FOR nIdxScan := 1 TO nNumberOfSensors DO
	//Setup parameters
		//Setup Motion part of sensor (Instance 0)
		arrNiko_P46xx[nIdxScan].eEventPriorityOccupancy:= stSensorSetup.eEventPriorityOccupancy;
		arrNiko_P46xx[nIdxScan].nHoldTimerOccupancy := stSensorSetup.nHoldTimerOccupancy ;
		arrNiko_P46xx[nIdxScan].nReportTimerOccupancy := stSensorSetup.nReportTimerOccupancy;
		arrNiko_P46xx[nIdxScan].nDeadtimeTimerOccupancy:= stSensorSetup.nDeadtimeTimerOccupancy;
		arrNiko_P46xx[nIdxScan].nSensitivityOccupancyA:= stSensorSetup.nSensitivityPIRSegmentA;
		arrNiko_P46xx[nIdxScan].nSensitivityOccupancyB:= stSensorSetup.nSensitivityPIRSegmentB;
		arrNiko_P46xx[nIdxScan].nSensitivityOccupancyC:= stSensorSetup.nSensitivityPIRSegmentC;
	
		//Setup Brightness part of sensor (Instance 1)
		arrNiko_P46xx[nIdxScan].bEnableBrightness := stSensorSetup.bEnableInstanceBrightness;
		arrNiko_P46xx[nIdxScan].eEventPriorityBrightness:= stSensorSetup.eEventPriorityBrightness;
		arrNiko_P46xx[nIdxScan].nDeadtimeTimerBrightness:= stSensorSetup.nDeadtimeTimerBrightness;
		arrNiko_P46xx[nIdxScan].nHysteresisBrightness:= stSensorSetup.nHysteresisBrightness;
		arrNiko_P46xx[nIdxScan].nHysteresisMinBrightness:= stSensorSetup.nHysteresisMinBrightness;
		arrNiko_P46xx[nIdxScan].nReportTimerBrightness:= stSensorSetup.nReportTimerBrightness;
		
	//Calculate delay time for init sensor
	arrtDelayTime[nIdxScan] := INT_TO_TIME((BYTE_TO_INT(arrShrtAdr[nIdxScan]) * 400));	
	arrDelaySetupDALIDevice[nIdxScan](IN:= bInitialize , PT:=arrtDelayTime[nIdxScan] , Q=> , ET=> );	
		
	IF arrDelaySetupDALIDevice[nIdxScan].q AND NOT GVL_DALI.arrbBlockDTR[DALI_LINE_NUM] AND NOT (arrInitDone[nIdxScan] OR arrInitErr[nIdxScan]) THEN
		arrInitSensor[nIdxScan]:= TRUE;
		GVL_DALI.arrbBlockDTR[DALI_LINE_NUM]:= TRUE;
	END_IF
	
	bQueryBrightness:= stPirSensorData.bQueryBrightness OR NOT bAutoRead;
	
	fbAutoRequestBrightness_TON(IN:= NOT fbAutoRequestBrightness_TON.Q  AND NOT stPirSensorData.bQueryBrightness , PT:= (arrtDelayTime[nIdxScan] + T#12M) , Q=>bAutoRead , ET=> );
	
	bQueryOccupancy:= NOT bAutoRead OR stPirSensorData.bQueryBrightness;
	
	arrNiko_P46xx[nIdxScan](
		bError=> , 
		ipResultMessage=> , 
		bInitialize:=  arrInitSensor[nIdxScan], 
		nShortAddress:= arrShrtAdr[nIdxScan], 
		nOptions:= , 
		bQueryOccupancy:= bQueryOccupancy, 
		bQueryBrightness:= bQueryBrightness, 
		bCancelHoldTimerOccupancy:= bCancelHoldTimerOccupancy, 
		bInitializing=> arrInitializing[nIdxScan] , 
		bReadingOccupancy=> , 
		bReadingBrightness=> , 
		bOccupied=> , 
		nBrightnessLevel=> );
	
	IF arrNiko_P46xx[nIdxScan].bError THEN
		GVL_DALI_LatestError.arrLineShrtAddr[DALI_LINE_NUM] :=arrShrtAdr[nIdxScan];
	END_IF
	
	arrInitDone_FTrig[nIdxScan](CLK:=arrInitializing[nIdxScan] );	
		IF arrInitDone_FTrig[nIdxScan].Q THEN
			IF NOT bInitTimeOut THEN
				arrInitDone[nIdxScan] := TRUE;
				GVL_DALI.arrbBlockDTR[DALI_LINE_NUM]:= FALSE;
			ELSE
				arrInitErr[nIdxScan] := TRUE;
				GVL_DALI.arrbBlockDTR[DALI_LINE_NUM]:= FALSE;
			END_IF
		END_IF
		
	fbInitTimeOut[nIdxScan](IN:=arrInitSensor[nIdxScan] AND NOT arrInitDone[nIdxScan], PT:= T#10S); 
	
	IF fbInitTimeOut[nIdxScan].Q THEN
		arrInitErr[nIdxScan] := TRUE;
		GVL_DALI.arrbBlockDTR[DALI_LINE_NUM]:= FALSE;
	END_IF
END_FOR

stPirSensorData.bPrc:= FALSE;
FOR nPirIdxOn:= 1 TO nNumberOfSensors DO
	IF arrNiko_P46xx[nPirIdxOn].bOccupied THEN
		stPirSensorData.bPrc:= TRUE;
		EXIT;
	END_IF
END_FOR

stPirSensorData.bBrightnessRead:=	arrNiko_P46xx[1].bReadingBrightness OR arrNiko_P46xx[2].bReadingBrightness OR arrNiko_P46xx[3].bReadingBrightness OR arrNiko_P46xx[4].bReadingBrightness OR arrNiko_P46xx[5].bReadingBrightness OR
														arrNiko_P46xx[6].bReadingBrightness OR arrNiko_P46xx[7].bReadingBrightness OR arrNiko_P46xx[8].bReadingBrightness OR arrNiko_P46xx[9].bReadingBrightness;

fBrightness_1:= F_fScale(0, arrSensorScales[1].fReadMaxSensor, 0, arrSensorScales[1].fMeassureMaxSensor, 0, arrNiko_P46xx[1].nBrightnessLevel);
fBrightness_2:= F_fScale(0, arrSensorScales[2].fReadMaxSensor, 0, arrSensorScales[2].fMeassureMaxSensor, 0, arrNiko_P46xx[2].nBrightnessLevel);
fBrightness_3:= F_fScale(0, arrSensorScales[3].fReadMaxSensor, 0, arrSensorScales[3].fMeassureMaxSensor, 0, arrNiko_P46xx[3].nBrightnessLevel);
fBrightness_4:= F_fScale(0, arrSensorScales[4].fReadMaxSensor, 0, arrSensorScales[4].fMeassureMaxSensor, 0, arrNiko_P46xx[4].nBrightnessLevel);
fBrightness_5:= F_fScale(0, arrSensorScales[5].fReadMaxSensor, 0, arrSensorScales[5].fMeassureMaxSensor, 0, arrNiko_P46xx[5].nBrightnessLevel);
fBrightness_6:= F_fScale(0, arrSensorScales[6].fReadMaxSensor, 0, arrSensorScales[6].fMeassureMaxSensor, 0, arrNiko_P46xx[6].nBrightnessLevel);
fBrightness_7:= F_fScale(0, arrSensorScales[7].fReadMaxSensor, 0, arrSensorScales[7].fMeassureMaxSensor, 0, arrNiko_P46xx[7].nBrightnessLevel);
fBrightness_8:= F_fScale(0, arrSensorScales[8].fReadMaxSensor, 0, arrSensorScales[8].fMeassureMaxSensor, 0, arrNiko_P46xx[8].nBrightnessLevel);
fBrightness_9:= F_fScale(0, arrSensorScales[9].fReadMaxSensor, 0, arrSensorScales[9].fMeassureMaxSensor, 0, arrNiko_P46xx[9].nBrightnessLevel);

IF fBrightness_1 <> 0 THEN
	stPirSensorData.fBrightness:= fBrightness_1;
END_IF
IF fBrightness_2 <> 0 THEN
	stPirSensorData.fBrightness:= MIN(fBrightness_2, stPirSensorData.fBrightness);
END_IF
IF fBrightness_3 <> 0 THEN
	stPirSensorData.fBrightness:=  MIN(fBrightness_3, stPirSensorData.fBrightness);
END_IF
IF fBrightness_4 <> 0 THEN
	stPirSensorData.fBrightness:=  MIN(fBrightness_4, stPirSensorData.fBrightness);
END_IF
IF fBrightness_5 <> 0 THEN
	stPirSensorData.fBrightness:=  MIN(fBrightness_5, stPirSensorData.fBrightness);
END_IF
IF fBrightness_6 <> 0 THEN
	stPirSensorData.fBrightness:= MIN(fBrightness_6, stPirSensorData.fBrightness);
END_IF
IF fBrightness_7 <> 0 THEN
	stPirSensorData.fBrightness:=  MIN(fBrightness_7, stPirSensorData.fBrightness);
END_IF
IF fBrightness_8 <> 0 THEN
	stPirSensorData.fBrightness:=  MIN(fBrightness_8, stPirSensorData.fBrightness);
END_IF
IF fBrightness_9 <> 0 THEN
	stPirSensorData.fBrightness:=  MIN(fBrightness_9, stPirSensorData.fBrightness);
END_IF


IF NOT bInitialize THEN
	FOR nIdxScan := 1 TO nNumberOfSensors DO
		fbInitTimeOut[nIdxScan](IN:= FALSE);
		arrInitDone[nIdxScan] := FALSE;
		arrInitErr[nIdxScan] := FALSE;
	END_FOR
END_IF
END_ACTION

END_FUNCTION_BLOCK

// POUs/DALI/FBs/FB_Short
FUNCTION_BLOCK INTERNAL FB_Short
VAR_INPUT
END_VAR
VAR_OUTPUT
END_VAR
VAR
END_VAR

END_FUNCTION_BLOCK

// POUs/DALI/FBs/FB_ValTrig_F
FUNCTION_BLOCK FB_ValTrig_F
VAR_INPUT
END_VAR
VAR_OUTPUT
END_VAR
VAR
END_VAR

END_FUNCTION_BLOCK

// POUs/DALI/FUNs/F_lrScale_EX
FUNCTION F_lrScale_EX : LREAL
VAR_INPUT
	fX0, fX1, fY0, fY1, fOffset : REAL;
	lrSetValDct					: REAL;
	bEnaLim 					: BOOL;
END_VAR
VAR
	fDeltaY						: REAL;
	fDeltaX						: REAL;
END_VAR

fDeltaY:= fY1-fY0;
fDeltaX :=fX1-fX0;

IF fDeltaX <=0 THEN
	fDeltaX:=1;
END_IF

IF bEnaLim THEN
	F_lrScale_EX:= LIMIT(fY0, REAL_TO_LREAL( (fDeltaY / fDeltaX) * lrSetValDct + fOffset), fY1);
ELSE
	F_lrScale_EX:= REAL_TO_LREAL( (fDeltaY / fDeltaX) * lrSetValDct + fOffset);
END_IF

END_FUNCTION

// POUs/DALI/MUX/Timing/FB_MinOnMinOffTime
FUNCTION_BLOCK  FB_MinOnMinOffTime
VAR
	nIdx: INT;
	fbTon: TON;
END_VAR
VAR_INPUT
	bRunCMD: BOOL;
	bStopCMD : BOOL;
	tMinOnTime: TIME;
	tMinOffTime: TIME;
END_VAR
VAR_OUTPUT
	bOut_Run: BOOL;
	bOut_Stop: BOOL;
END_VAR

CASE nIdx OF

0: (*Init Step*)

bOut_Run:= FALSE;
bOut_Stop:= FALSE;
fbTon(IN:=FALSE);

IF bRunCMD THEN
	nIdx := nIdx + 1;
END_IF

1: (*Check min on Time*)

fbTon(IN:= TRUE, PT:= tMinOnTime , Q=> , ET=> );
bOut_Run:= TRUE;

IF fbTon.Q THEN
	nIdx := nIdx + 1;
END_IF

2: (*Kørsel OK*)

fbTon(IN:= FALSE);

IF bStopCMD THEN
	bOut_Stop:= TRUE;
	bOut_Run:= FALSE;
	nIdx := nIdx + 1;
END_IF

3: (*Check Min Off tiden*)

fbTon(IN:= TRUE, PT:= tMinOffTime , Q=> , ET=> );

IF fbTon.Q THEN
	nIdx := 0;
END_IF






















ELSE
	nIdx := 0;

END_CASE

END_FUNCTION_BLOCK

// POUs/DALI/Operators/FB_BA_Swi
FUNCTION_BLOCK FB_BA_Swi
VAR_INPUT
	bOn : BOOL;
	bOff : BOOL;
	bToggle : BOOL;
END_VAR
VAR_OUTPUT
	bLgt: BOOL;
END_VAR
VAR
	fbOn_RTrig: R_TRIG;
	fbOff_RTrig: R_TRIG;
	fbTogle_RTrig: R_TRIG;

END_VAR


fbOn_RTrig(CLK:= bOn );
fbOff_RTrig(CLK:= bOn );
fbTogle_RTrig(CLK:= bOn );

IF fbOn_RTrig.Q THEN
	bLgt := TRUE;
END_IF

IF fbOff_RTrig.Q THEN
	bLgt := FALSE;
END_IF

IF fbTogle_RTrig.Q THEN
	bLgt := NOT bLgt;
END_IF

END_FUNCTION_BLOCK

// POUs/DALI/Operators/FB_Click
FUNCTION_BLOCK FB_Click
VAR_INPUT
	bSwitch						:	BOOL; (* Input signal. *)
	tSwitchTime					:	TIME := T#50MS; (* Kontrol af længde på tryk *)
END_VAR
VAR_OUTPUT
	bShortClick					:	BOOL; (* Kort tryk indikering *)
	bLongClick					:	BOOL; (* Lang tryk indikering *)
END_VAR
VAR
	fbTimerDelay_TON			:	TON;
	fbRisingEdgeSwitch			:	R_TRIG;
	fbFallingEdgeSwitch			:	F_TRIG;
	bDelayOver					:	BOOL := FALSE;
END_VAR

bShortClick := FALSE;
bLongClick := FALSE;

fbRisingEdgeSwitch(CLK := bSwitch);
IF (fbRisingEdgeSwitch.Q) THEN
	fbTimerDelay_TON(IN := FALSE);
	bDelayOver := FALSE;
END_IF

fbFallingEdgeSwitch(CLK := bSwitch);
IF (fbFallingEdgeSwitch.Q) THEN
	IF (NOT bDelayOver) THEN
		bShortClick := TRUE;
		bLongClick := FALSE;
	END_IF
END_IF

IF (bSwitch AND NOT bDelayOver) THEN
	fbTimerDelay_TON(IN := TRUE, PT := tSwitchTime);
	IF (fbTimerDelay_TON.Q) THEN
		fbTimerDelay_TON(IN := FALSE);
		bDelayOver := TRUE;
		bShortClick := FALSE;
		bLongClick := TRUE;
	END_IF
END_IF

END_FUNCTION_BLOCK

// POUs/DALI/Operators/FB_FileCopy
FUNCTION_BLOCK FB_FileCopy
VAR_INPUT
	srcNetId			: T_AmsNetId;	(* TwinCAT network address of the source file *)
	srcFileName			: T_MaxString;	(* source file path and name *)
	destNetId			: T_AmsNetId;	(* TwinCAT network address of the destination file *)
	destFileName		: T_MaxString;  (* destination file path and name *)
	bExecute			: BOOL;			(* rising edge start fb execution *)
	tAdsTimeOut			: TIME;			(* ads timeout *)
END_VAR
VAR_OUTPUT
	bBusy				:BOOL;
	bError				:BOOL;
	nErrId				:UDINT;
END_VAR
VAR
	fbFileOpen			:FB_FileOpen;
	fbFileClose			:FB_FileClose;
	fbFileRead			:FB_FileRead;
	fbFileWrite			:FB_FileWrite;

	hSrcFile			:UINT	:= 0;(* file handle of the source file *)
	hDestFile			:UINT	:= 0;(* file handle of the destination file *)

	Step				:DWORD;
	RisingEdge			:R_TRIG;

	buffRead			:ARRAY[1..9999] OF BYTE;(* buffer *)
	cbReadLength		:UDINT:=0;
END_VAR

RisingEdge(CLK:=bExecute);
IF RisingEdge.Q THEN
	IF NOT bBusy THEN
		bBusy := TRUE;
		bError:= FALSE;
		nErrId:=0;
		Step := 1;
		cbReadLength:=0;
		hSrcFile:=0;
		hDestFile:=0;
	END_IF
END_IF


CASE Step OF
	0:	(* do nothing *)
		;

	1:	(* open source file *)
		fbFileOpen(  bExecute := FALSE  );
		fbFileOpen( 	sNetId := srcNetId,
						sPathName := srcFileName,
						nMode := FOPEN_MODEREAD OR FOPEN_MODEBINARY,
						ePath := PATH_GENERIC,
						tTimeout := tAdsTimeout,
						bExecute := TRUE );
		Step := Step + 1;

	2:
		fbFileOpen( bExecute := FALSE );
		IF ( NOT fbFileOpen.bBusy ) THEN
			IF ( fbFileOpen.bError ) THEN
				nErrId := fbFileOpen.nErrId;
				bError := TRUE;
				Step := 50;
			ELSE
				hSrcFile := fbFileOpen.hFile;
				Step := Step + 1;
			END_IF
		END_IF

	3:	(* open destination file *)
		fbFileOpen(  bExecute := FALSE  );
		fbFileOpen( 	sNetId := destNetId,
						sPathName := destFileName,
						nMode := FOPEN_MODEWRITE OR FOPEN_MODEBINARY,
						ePath := PATH_GENERIC,
						tTimeout := tAdsTimeout,
						bExecute := TRUE );
		Step := Step+1;

	4:
		fbFileOpen(  bExecute := FALSE  );
		IF ( NOT fbFileOpen.bBusy ) THEN
			IF ( fbFileOpen.bError ) THEN
				nErrId := fbFileOpen.nErrId;
				bError := TRUE;
				Step := 50;
			ELSE
				hDestFile := fbFileOpen.hFile;
				Step := Step + 1;
			END_IF
		END_IF

	5:	(*read data from source file*)
		cbReadLength := 0;
		fbFileRead( bExecute:= FALSE );
		fbFileRead( 	sNetId:=SrcNetId,
						hFile:=hSrcFile,
						pReadBuff:= ADR(buffRead),
						cbReadLen:= SIZEOF(buffRead),
						bExecute:=TRUE,
						tTimeout:=tAdsTimeOut );
		Step := Step + 1;

	6:
		fbFileRead( bExecute:= FALSE );
		IF ( NOT fbFileRead.bBusy ) THEN
			IF ( fbFileRead.bError ) THEN
				nErrId := fbFileRead.nErrId;
				bError := TRUE;
				Step := 50;
			ELSE
				cbReadLength := fbFileRead.cbRead;
				Step := Step + 1;
			END_IF
		END_IF

	7:	(*write data to destination file*)
		fbFileWrite( bExecute := FALSE );
		fbFileWrite(	sNetId:=DestNetId,
						hFile:=hDestFile,
						pWriteBuff:= ADR(buffRead),
						cbWriteLen:= cbReadLength,
						bExecute:=TRUE,
						tTimeout:=tAdsTimeOut );
		Step := Step + 1;

	8:
		fbFileWrite( bExecute := FALSE );
		IF ( NOT fbFileWrite.bBusy ) THEN
			IF ( fbFileWrite.bError ) THEN
				nErrId := fbFileWrite.nErrId;
				bError := TRUE;
				Step := 50;
			ELSE
				IF fbFileRead.bEOF THEN (*Check if the EOF flag ist set *)
					Step := 50;		(*cleanup: close the destination and source files *)
				ELSE
					Step := 5; (* repeat reading *)
				END_IF
			END_IF
		END_IF

	30:	(* close the destination file *)
		fbFileClose( bExecute := FALSE );
		fbFileClose( 	sNetId:=destNetId,
						hFile:=hDestFile,
						bExecute:=TRUE,
						tTimeout:=tAdsTimeOut );
		Step := Step + 1;

	31:
		fbFileClose( bExecute := FALSE );
		IF ( NOT fbFileClose.bBusy ) THEN
			IF ( fbFileClose.bError ) THEN
				nErrId := fbFileClose.nErrId;
				bError := TRUE;
			END_IF
			Step := 50;
			hDestFile := 0;
		END_IF

	40: (* close source file *)
		fbFileClose( bExecute := FALSE );
		fbFileClose( 	sNetId:=srcNetId,
						hFile:=hSrcFile,
						bExecute:=TRUE,
						tTimeout:=tAdsTimeOut );
		Step := Step + 1;

	41:
		fbFileClose( bExecute := FALSE );
		IF ( NOT fbFileClose.bBusy ) THEN
			IF ( fbFileClose.bError ) THEN
				nErrId := fbFileClose.nErrId;
				bError := TRUE;
			END_IF
			Step := 50;
			hSrcFile := 0;
		END_IF

	50: (*error or ready => cleanup*)
		IF ( hDestFile <> 0 ) THEN
			Step := 30; (* close the destination file*)
		ELSIF (hSrcFile <> 0 ) THEN
			Step := 40; (* close the source file *)
		ELSE
			Step := 0;	(* ready *)
			bBusy := FALSE;
		END_IF

END_CASE

END_FUNCTION_BLOCK

// POUs/DALI/Operators/FB_Ramper
FUNCTION_BLOCK FB_Ramper
VAR_INPUT
	bEnable							:	BOOL; (* A positive input enables the function block. A negative state deactivates the inputs and sets the function-block to the idle-mode. *)
	bOn								:	BOOL; (* A rising edge sets the output nLightLevel directly to the maximum-level (32767). *)
	bOff							:	BOOL; (* A rising edge sets the output nLightLevel immediately to "0". *)
	bToggle							:	BOOL; (* Rising edges at this input toggle the nLightLevel between "0" and "32767". *)
	bStart							:	BOOL; (* This input starts the dim-ramp from the actual value to nEndLevel within the time defined as tRampTime. This can be interrupted by bOn, bOff or bToggle at any time. *)
	nEndLevel						:	INT; (* Target-value of the dim-ramp. *)
	tRampTime						:	TIME := t#10s; (* Ramp-time, see bStart. (initial value: 10s). *)
	nOptions						:	DWORD; (* Reserved for future developments. *)
END_VAR
VAR_OUTPUT
	bLight							:	BOOL; (* As long as nLightLevel is greater than "0", this output is set to TRUE. *)
	bBusy							:	BOOL; (* When the block is activated the output is set, and it remains active until execution of the command has been completed. *)
	bError							:	BOOL; (* This output is switched to TRUE if an error occurs during the execution of a command. The command-specific error code is contained in nErrorId. bError is reset to FALSE by the execution of an instruction at the inputs. *)
	nErrorId						:	UDINT; (* Contains the command-specific error code of the most recently executed command. nErrorId is reset to 0 by the execution of an instruction at the inputs. See Error codes. *)
END_VAR
VAR_IN_OUT
	nLightLevel						:	INT; (* Reference to the actual light-level-output. This output has to be an IN-OUT-Variable because the function-block may need the actual level as a start-level for a ramp. *)
END_VAR
VAR
	fbRTrigEnable					:	R_TRIG;
	fbRTrigOn						:	R_TRIG;
	fbRTrigOff						:	R_TRIG;
	fbRTrigToggle					:	R_TRIG;
	fbRTrigStart					:	R_TRIG;
	nStep							:	INT;
	fbTonRamp						:	TON;
	tRampTime_M						:	TIME;
	fLightLevel						:	LREAL;
	fStartLevel						:	LREAL;
	fEndLevel_M						:	LREAL;
	nEndLevel_M						:	INT;
	bOffCmdPreset					:	BOOL;
	bOnCmdPreset					:	BOOL;
	bToggleCmdPreset				:	BOOL;
	bStartCmdPreset					:	BOOL;

	(*For test-purposes*)
	nSetpointValue					:	INT;	(*for scope-purposes only*)
END_VAR

fbRTrigEnable(CLK := bEnable);
IF (fbRTrigEnable.Q) THEN
	bBusy := FALSE;
	nErrorId := 0;
	bError := FALSE;
END_IF


(*Start-conditions*)
fbRTrigOn(CLK := bOn);
IF (fbRTrigOn.Q AND bEnable) THEN
	bOnCmdPreset := TRUE;
END_IF
fbRTrigOff(CLK := bOff);
IF (fbRTrigOff.Q AND bEnable) THEN
	bOffCmdPreset := TRUE;
END_IF
fbRTrigToggle(CLK := bToggle);
IF (fbRTrigToggle.Q AND bEnable) THEN
	bToggleCmdPreset := TRUE;
END_IF
fbRTrigStart(CLK := bStart);
IF (fbRTrigStart.Q AND bEnable AND NOT bBusy) THEN
	bStartCmdPreset := TRUE;
END_IF

CASE nStep OF
0:
	bBusy := FALSE;

	IF (bOnCmdPreset) THEN
		bOnCmdPreset := FALSE;
		bBusy := TRUE;
		nErrorId := 0;
		bError := FALSE;
		nStep := 10;
	END_IF
	IF (bOffCmdPreset) THEN
		bOffCmdPreset := FALSE;
		bBusy := TRUE;
		nErrorId := 0;
		bError := FALSE;
		nStep := 15;
	END_IF
	IF (bToggleCmdPreset) THEN
		bToggleCmdPreset := FALSE;
		bBusy := TRUE;
		nErrorId := 0;
		bError := FALSE;
		nStep := 5;
	END_IF
	IF (bStartCmdPreset) THEN
		bStartCmdPreset := FALSE;
		bBusy := TRUE;
		nErrorId := 0;
		bError := FALSE;
		nStep := 20;
	END_IF

	
(*-----------------------------------------------------------------------------------*)
(*Toggle-decision*)

5:	IF bLight THEN
		nStep := 15;
	ELSE
		nStep := 10;
	END_IF


(*-----------------------------------------------------------------------------------*)
(*On*)

10:	
	nLightLevel :=32767;			
	nSetpointValue:=nLightLevel;
	nStep := 0;

(*-----------------------------------------------------------------------------------*)
(*Off*)

15:
	nLightLevel :=0;
	nSetpointValue:=nLightLevel;
	nStep := 0;


(*-----------------------------------------------------------------------------------*)
(*Ramp-driving*)


20:	
	tRampTime_M := tRampTime;
	nEndLevel_M := nEndLevel;
	fEndLevel_M := INT_TO_LREAL(nEndLevel_M);
	fStartLevel	:= INT_TO_LREAL(nLightLevel);
	fbTonRamp(IN:=FALSE);
	fbTonRamp(IN:=TRUE,PT:=tRampTime);
	nStep := 50;

	nSetpointValue:=nEndLevel_M;


(*BEGIN LOOP*)

50:	
	fbTonRamp();

	IF (tRampTime_M > t#0s) THEN
		fLightLevel := fStartLevel + (((fEndLevel_M-fStartLevel)/TIME_TO_LREAL(tRampTime_M))*TIME_TO_LREAL(fbTonRamp.ET));
		nLightLevel := ABS(LREAL_TO_INT(fLightLevel));
	ELSIF (tRampTime_M = t#0s) THEN
		nLightLevel := nEndLevel_M;
	END_IF


	IF (nLightLevel = nEndLevel_M) THEN
		nStep := 0;
	ELSE
		nStep := 100;
	END_IF

100:
	IF (bEnable) THEN
		nStep := 50;
		IF (bToggleCmdPreset) THEN
			bToggleCmdPreset := FALSE;
			nStep := 5;
		END_IF
		IF (bOnCmdPreset) THEN
			bOnCmdPreset := FALSE;
			nStep := 10;
		END_IF
		IF (bOffCmdPreset) THEN
			bOffCmdPreset := FALSE;
			nStep := 15;
		END_IF
	ELSE
		nStep := 0;
	END_IF

END_CASE

bLight := nLightLevel>0;

END_FUNCTION_BLOCK

// POUs/DALI/Power Control/FB_AutoTune_TcBA_EX
FUNCTION_BLOCK FB_AutoTune_TcBA_EX
VAR
	nTuneStep : INT;
	fbDelayTune_TON:TON;
	fbTimeOutStep_TON:TON;

	iStepBeforeError: INT;
	fbR_TrigRunTuning: R_TRIG;
	nTuneIdx: INT := 0;
END_VAR
VAR_INPUT
	bRunTuning: BOOL;
	tTuningDelay:TIME:=T#10S;
END_VAR
VAR_OUTPUT
	bTuningInProcess: BOOL;
	sActProcess: STRING;
	bTuningDone: BOOL;
	bSetValDct: BOOL;
	fSetValDct: REAL;
END_VAR
VAR_IN_OUT PERSISTENT
	
END_VAR
VAR_IN_OUT
	stTuneData			: ST_TuneData_EX;
	stPirSensorData		: ST_DALI_Sensor;
END_VAR

bTuningDone:=stTuneData.bTunnigDone;

CASE nTuneStep OF

0: (*Init step*)

	sActProcess:='Waiting for command';

	bSetValDct:=FALSE;
	fSetValDct:=0;

	bTuningInProcess:= FALSE;
	fbDelayTune_TON(IN:=FALSE);
	fbTimeOutStep_TON(IN:=FALSE, PT:=T#1S);

	fbR_TrigRunTuning(CLK:= bRunTuning, Q=> );

	IF fbR_TrigRunTuning.Q THEN
		nTuneIdx:=0;
		bTuningInProcess:= TRUE;
		bTuningDone:=FALSE;
		stTuneData.bTunnigDone:=FALSE;
		nTuneStep:= nTuneStep +1;
		stPirSensorData.bQueryBrightness:= FALSE;
		sActProcess:='Testing 1%';
		fSetValDct:= 1 ;
	END_IF

1: 	(*Test xx% to group*)

	bSetValDct:=TRUE ;

	IF bSetValDct THEN
		stPirSensorData.bQueryBrightness:= FALSE;
		nTuneStep:= nTuneStep +1;
	END_IF

2:	(*Check if call are done correcly*)
	bSetValDct:=FALSE;
	
	(* Done *)
	fbDelayTune_TON(IN:= TRUE , PT:= tTuningDelay);
		IF fbDelayTune_TON.Q THEN
			stPirSensorData.bQueryBrightness:= TRUE;
			nTuneStep:= 3;
		END_IF
	
3:
	fbTimeOutStep_TON(IN:= TRUE);
	IF NOT fbTimeOutStep_TON.Q THEN
		IF stPirSensorData.bBrightnessRead THEN
			nTuneStep:= 10;
			bSetValDct:=FALSE ;
			stTuneData.arrLuxLevels[nTuneIdx]:=stPirSensorData.fBrightness;
			fbDelayTune_TON(IN:= FALSE);
			fbTimeOutStep_TON(IN:=FALSE);
			stPirSensorData.bQueryBrightness:= FALSE;
		END_IF
	ELSE
		nTuneStep:= 999;
	END_IF

10:
	IF nTuneIdx <= 20 THEN
		nTuneIdx:=nTuneIdx + 1;
		nTuneStep:= 1;
		sActProcess:= CONCAT('Testing ', INT_TO_STRING(nTuneIdx*5));
		sActProcess:= CONCAT(sActProcess, '%');
		fSetValDct:= nTuneIdx*5 ;
	ELSE
		nTuneStep:= 888;
	END_IF

888:	(* Tuning Data success*)
	nTuneStep:=0;
	bRunTuning:=FALSE;
	bTuningDone:=TRUE;
	fSetValDct:= 0 ;
	bSetValDct:=TRUE ;
	stTuneData.bTunnigDone:=TRUE;

	fbTimeOutStep_TON(IN:= TRUE, PT:= T#1s);
	IF fbTimeOutStep_TON.Q THEN
		stPirSensorData.bQueryBrightness:= FALSE;
		nTuneStep:= 0;
	END_IF


999:	(* Error *)

		bRunTuning:=FALSE;
		fbTimeOutStep_TON(IN:= TRUE, PT:= T#1s);
		IF fbTimeOutStep_TON.Q THEN
			stPirSensorData.bQueryBrightness:= FALSE;
			nTuneStep:= 0;
		END_IF
ELSE
	nTuneStep:=0;
END_CASE

END_FUNCTION_BLOCK

// POUs/DALI/Power Control/FB_DirectLight_1Group
FUNCTION_BLOCK FB_DirectLight_1Group
VAR_INPUT
	_bEnable:BOOL;
	_bSyncVal:BOOL;
	_fSyncVal:REAL;
	_fSP : REAL;
	_bTuningInProcess: BOOL;
	_bSetValDct: BOOL;
	_fSetValDct: REAL;
	_bDimUp : BOOL;
	_bDimDown : BOOL;
	_bOff : BOOL;
	_fActlLgtLvl: REAL;
	_bRecallManualLevel: BOOL;
END_VAR
VAR_OUTPUT
	fSP_Group	: REAL;
	bWriteValue : BOOL;
	bDimUp : BOOL;
	bDimDwn : BOOL;
	bOff : BOOL;
	bClMinCtrlVal: BOOL;
END_VAR
VAR_IN_OUT
	stPirSensorData		: ST_DALI_Sensor;
END_VAR
VAR
	lrDiff: REAL;
	lrDiffPct:REAL;
	fbStepTimer_TON: TON;
	lrDiffAbs: REAL;
	bDoNothing: BOOL;

	fbStartUpVal: R_TRIG;
	fbStartUp: R_TRIG;

	fbF_Trig: F_TRIG;
	_fSPOld: REAL;
	
	fbTurnOff: R_TRIG;
	fbRTrig_DataRead: R_TRIG;
	fbReadLiveValue_TON :TON ;	
	fbCheckReadBrightness: TON;

	tCycleTimer: TIME;
	fbResendWrieteValue_TON: TON;
END_VAR

//New data from sensor
fbRTrig_DataRead(CLK:= stPirSensorData.bBrightnessRead);

//Checking the Read aren't keept high for long periode
fbCheckReadBrightness(IN:= stPirSensorData.bQueryBrightness , PT:= T#500MS , Q=> , ET=> );

IF fbCheckReadBrightness.Q OR fbRTrig_DataRead.Q THEN
	stPirSensorData.bQueryBrightness:= FALSE;
END_IF	

tCycleTimer:= SEL(_bEnable, T#1M, T#15S);

fbReadLiveValue_TON(IN:= NOT fbReadLiveValue_TON.Q, PT:= tCycleTimer, Q=> , ET=> );
IF fbReadLiveValue_TON.Q THEN
	stPirSensorData.bQueryBrightness := TRUE;
END_IF

bOff:= FALSE;
(*Lukker korrekt skrive bit, efter endt Tuning*)
	fbF_Trig(CLK:=_bTuningInProcess , Q=> );
	fbTurnOff(CLK:= (_fSP = 0) , Q=> );
	IF fbF_Trig.Q THEN
		bWriteValue:= FALSE;
	END_IF

IF NOT _bTuningInProcess THEN

	IF NOT _bEnable THEN
			IF _bDimUp THEN
				IF _fActlLgtLvl = 0 THEN
					bClMinCtrlVal := TRUE;
				ELSE
					bClMinCtrlVal := FALSE;
					bDimUp:= TRUE;
				END_IF
			ELSE
					bClMinCtrlVal := FALSE;
					bDimUp:= FALSE;
			END_IF

	IF _bOff OR fbTurnOff.Q THEN
		bOff:= TRUE;
		fSP_Group:= 0;
	END_IF
		bDimDwn:= _bDimDown;
		_fSPOld:=0;
	END_IF


	IF _fSP <> 0  AND _bEnable  THEN

		bWriteValue:= FALSE;

		IF _fSP <> _fSPOld THEN
			fSP_Group := _fSP;
			_fSPOld := _fSP;
			bWriteValue:= TRUE;
		END_IF
		
		fbResendWrieteValue_TON(IN:= (ABS(fSP_Group - _fActlLgtLvl) > 1) AND NOT fbResendWrieteValue_TON.Q, PT:= T#2S);
		IF fbResendWrieteValue_TON.Q THEN
			bWriteValue:= TRUE;
		END_IF
	END_IF	
ELSE
		fSP_Group:=_fSetValDct;
		bWriteValue:= _bSetValDct;
END_IF

IF _bRecallManualLevel THEN
		fSP_Group:=_fSetValDct;
		bWriteValue:= _bSetValDct;
END_IF

END_FUNCTION_BLOCK

// POUs/DALI/Power Control/FB_LightCtrl_1Group
FUNCTION_BLOCK FB_LightCtrl_1Group
VAR_INPUT
	_bEnable:BOOL;
	_bSyncVal:BOOL;
	_fSyncVal:REAL;
	_fSP : REAL;
	_fPV : REAL;
	_fStep1Limit: REAL;
	_fSPStep1 : REAL;
	_fStep2Limit: REAL;
	_fSPStep2 : REAL;
	_fStep3Limit: REAL;
	_fSPStep3 : REAL;
	_fStep4Limit: REAL;
	_fSPStep4 : REAL;
	_fStep5Limit: REAL;
	_fSPStep5 : REAL;
	_tStepTime : TIME;
	_bStepModeCalculationOnSP:BOOL;
	_bTuningInProcess: BOOL;
	_bSetValDct: BOOL;
	_fSetValDct: REAL;
	_bDimUp : BOOL;
	_bDimDown : BOOL;
	_bOff : BOOL;
	_fActlLgtLvl: REAL;
	_bRecallManualLevel: BOOL;
	_fMinOutputPowerLevel : REAL;
	_fMaxOutputPowerLevel : REAL;
END_VAR
VAR_OUTPUT
	fSP_Group	: REAL;
	bWriteValue : BOOL;
	bDimUp : BOOL;
	bDimDwn : BOOL;
	bOff : BOOL;
	bClMinCtrlVal: BOOL;
END_VAR
VAR_IN_OUT
	stPirSensorData		: ST_DALI_Sensor;
END_VAR
VAR
	fDiff: REAL;
	fDiffPct:REAL;
	fbStepTimer_TON: TON;
	fDiffAbs: REAL;
	bDoNothing: BOOL;
	bStep1: BOOL;
	bStep2: BOOL;
	bStep3: BOOL;
	bStep4: BOOL;
	bStep5: BOOL;
	bIncrease: BOOL;
	bDecrease: BOOL;
	fbStartUpVal: R_TRIG;
	fbStartUp: R_TRIG;
	fStepSize_1: REAL;
	fStepSize_2: REAL;
	fStepSize_3: REAL;
	fStepSize_4: REAL;
	fStepSize_5: REAL;
	fbTurnOff: R_TRIG;
	fbF_Trig: F_TRIG;
	fbBA_ValTrigf : FB_BA_ValTrigf;
	bTurnOff: BOOL;
	bWriteValueRTrig: BOOL;
	bActiveFB: BOOL;
	fbManFTRIG: F_TRIG;
	fHys: INT;
	fbRTrig_DataRead: R_TRIG;
	fbCheckOffValueDetect_TON: TON;
	fbTurnOffLight_TOF: TOF;
	fbBA_ValTrigLR : FB_BA_ValTrigF ;
	fbCheckCorrectLevel: TON;
	fbCheckReadBrightness: TON;
	fbDelayResend_TON: TON;
	bReSendCmd: BOOL;
	bEnableCtrl: BOOL;
	fbDelaysReleaseCtrl: TON;
END_VAR

//New data from sensor
fbRTrig_DataRead(CLK:= stPirSensorData.bBrightnessRead);

//Checking the Read aren't keept high for long periode
fbCheckReadBrightness(IN:= stPirSensorData.bQueryBrightness , PT:= T#500MS , Q=> , ET=> );

IF fbCheckReadBrightness.Q OR fbRTrig_DataRead.Q THEN
	stPirSensorData.bQueryBrightness:= FALSE;
END_IF

(*Beregninger for differencen mellem SP og PV*)
IF fbRTrig_DataRead.Q THEN
	fDiff:=_fSP-_fPV;
	fDiffAbs:= ABS(_fSP-_fPV);
	IF fDiffAbs >0 THEN
		IF _fsp<= 0 THEN
			fDiffPct:= 100;
		ELSE
			fDiffPct:= (fDiffAbs / _fSP )*100;
		END_IF
	END_IF

	(*Check if we need to lower or raise the output *)
	bIncrease:= FALSE;
	bDecrease:= FALSE;
	
	IF fDiff < 0 THEN
		bDecrease:= TRUE;
	ELSE
		bIncrease:= TRUE;
	END_IF
END_IF

//Continous calculating step size

bDoNothing:= FALSE;
bStep1:= FALSE;
bStep2:= FALSE;
bStep3:= FALSE;
bStep4:= FALSE;
bStep5:= FALSE;

IF _bStepModeCalculationOnSP THEN
	fStepSize_1:=_fSP * (_fSPStep1 / 100);
	fStepSize_2:=_fSP *( _fSPStep2 / 100);
	fStepSize_3:=_fSP *( _fSPStep3 / 100);
	fStepSize_4:=_fSP *( _fSPStep4 / 100);
	fStepSize_5:=_fSP *( _fSPStep5 / 100);
ELSE
	fStepSize_1:=_fSPStep1;
	fStepSize_2:=_fSPStep2;
	fStepSize_3:= _fSPStep3;
	fStepSize_4:= _fSPStep4;
	fStepSize_5:=_fSPStep5;
END_IF

IF fDiffPct <= _fStep1Limit THEN
	bDoNothing:= TRUE;
END_IF

IF (fDiffPct > _fStep1Limit) AND  (fDiffPct <= _fStep2Limit) THEN
	bStep1:= TRUE;
END_IF

IF (fDiffPct > _fStep2Limit) AND  (fDiffPct <= _fStep3Limit) THEN
	bStep2:= TRUE;
END_IF

IF (fDiffPct > _fStep3Limit) AND  (fDiffPct <= _fStep4Limit) THEN
	bStep3:= TRUE;
END_IF

IF (fDiffPct > _fStep4Limit) AND  (fDiffPct <= _fStep5Limit) THEN
	bStep4:= TRUE;
END_IF

IF (fDiffPct > _fStep5Limit)  THEN
	bStep5:= TRUE;
END_IF

//LightCtrlProcess
IF NOT _bTuningInProcess THEN
	IF NOT _bEnable THEN
		IF _bDimUp THEN
			IF _fActlLgtLvl = 0 THEN
				bClMinCtrlVal := TRUE;
			ELSE
				bClMinCtrlVal := FALSE;
				bDimUp:= TRUE;
			END_IF
		ELSE
				bClMinCtrlVal := FALSE;
				bDimUp:= FALSE;
		END_IF
		bDimDwn:= _bDimDown;

	END_IF

	IF _fSP <> 0  AND _bEnable  THEN
		fbTurnOff(CLK:= FALSE , Q=> );
		fbStepTimer_TON(IN:=_bEnable AND NOT fbStepTimer_TON.q , PT:=_tStepTime , Q=> , ET=> );
		
		fbDelaysReleaseCtrl(IN:= bEnableCtrl , PT:=T#5S , Q=> , ET=> );

		IF fbDelaysReleaseCtrl.Q THEN 

	 		IF fbStepTimer_TON.Q THEN
				stPirSensorData.bQueryBrightness := TRUE;
			END_IF

			(*Controlling the step rate*)
			IF (fbRTrig_DataRead.Q OR fbStartUp.Q) OR bTurnOff  THEN
				stPirSensorData.bQueryBrightness := FALSE;
				IF bStep1 THEN
					IF bDecrease THEN
						fSP_Group:=LIMIT (_fMinOutputPowerLevel, (fSP_Group - fStepSize_1), _fMaxOutputPowerLevel);
					END_IF
	
					IF bIncrease THEN
						fSP_Group:=LIMIT (_fMinOutputPowerLevel, (fSP_Group +  fStepSize_1), _fMaxOutputPowerLevel);
					END_IF
				END_IF
	
				IF bStep2 THEN
					IF bDecrease THEN
						fSP_Group:=LIMIT (_fMinOutputPowerLevel, (fSP_Group - fStepSize_2), _fMaxOutputPowerLevel);
					END_IF
	
					IF bIncrease THEN
						fSP_Group:=LIMIT (_fMinOutputPowerLevel, (fSP_Group +  fStepSize_2), _fMaxOutputPowerLevel);
					END_IF
				END_IF
	
				IF bStep3 THEN
					IF bDecrease THEN
						fSP_Group:=LIMIT (_fMinOutputPowerLevel, (fSP_Group - fStepSize_3), _fMaxOutputPowerLevel);
					END_IF
	
					IF bIncrease THEN
						fSP_Group:=LIMIT (_fMinOutputPowerLevel, (fSP_Group +  fStepSize_3), _fMaxOutputPowerLevel);
					END_IF
				END_IF
	
				IF bStep4 THEN
					IF bDecrease THEN
						fSP_Group:=LIMIT (_fMinOutputPowerLevel, (fSP_Group - fStepSize_4), _fMaxOutputPowerLevel);
					END_IF
	
					IF bIncrease THEN
						fSP_Group:=LIMIT (_fMinOutputPowerLevel, (fSP_Group +  fStepSize_4), _fMaxOutputPowerLevel);
					END_IF
				END_IF
	
				IF bStep5 THEN
					IF bDecrease THEN
						fSP_Group:=LIMIT (_fMinOutputPowerLevel, (fSP_Group - fStepSize_5), _fMaxOutputPowerLevel);
					END_IF
	
					IF bIncrease THEN
						fSP_Group:=LIMIT (_fMinOutputPowerLevel, (fSP_Group +  fStepSize_5), _fMaxOutputPowerLevel);
					END_IF
				END_IF
			END_IF
		END_IF
		
	ELSE
		fSP_Group := 0;
	END_IF


ELSE
	fSP_Group:=_fSetValDct;
	bWriteValue:= _bSetValDct;
END_IF

fbStartUpVal(CLK:=_bSyncVal , Q=> );

IF fbStartUpVal.Q THEN
	fSP_Group:= LIMIT(_fMinOutputPowerLevel, _fSyncVal, _fMaxOutputPowerLevel);
	bEnableCtrl:= TRUE;
END_IF

IF _bRecallManualLevel THEN
		fSP_Group:=_fSetValDct;
		bWriteValue:= _bSetValDct;
END_IF

(*Lukker korrekt skrive bit, efter endt Tuning*)
	fbF_Trig(CLK:=_bTuningInProcess , Q=> );

	IF fbF_Trig.Q THEN
		bWriteValue:= FALSE;
	END_IF


fbTurnOff(CLK:= _fSP = 0 , Q=> );

IF (ABS(_fActlLgtLvl - fSP_Group) > 2)  AND _bEnable THEN
	fbDelayResend_TON(IN:=TRUE , PT:= T#15S, Q=> , ET=> );
	IF fbDelayResend_TON.Q THEN
		bReSendCmd:= TRUE;
		fbDelayResend_TON(IN:=FALSE);
	ELSE
		bReSendCmd:= FALSE;
	END_IF
END_IF

fbBA_ValTrigf(
	bEn:=TRUE ,
	bRetrig:= _bOff OR fbTurnOff.Q OR bReSendCmd,
	fIn:= fSP_Group ,
	fHys:=0.5,
	fOut=> ,
	bSet=>bWriteValue);

END_FUNCTION_BLOCK

// POUs/DALI/Power Control/FB_LightCtrl_1Group_
FUNCTION_BLOCK FB_LightCtrl_1Group_
VAR_INPUT
	_bEnable:BOOL;
	_bSyncVal:BOOL;
	_fSyncVal:REAL;
	_fSP : REAL;
	_fPV : REAL;
	_fStep1Limit: REAL;
	_fSPStep1 : REAL;
	_fStep2Limit: REAL;
	_fSPStep2 : REAL;
	_fStep3Limit: REAL;
	_fSPStep3 : REAL;
	_fStep4Limit: REAL;
	_fSPStep4 : REAL;
	_fStep5Limit: REAL;
	_fSPStep5 : REAL;
	_tStepTime : TIME;
	_bStepModeCalculationOnSP:BOOL;
	_bTuningInProcess: BOOL;
	_bSetValDct: BOOL;
	_fSetValDct: REAL;
	_bDimUp : BOOL;
	_bDimDown : BOOL;
	_bOff : BOOL;
	_fActlLgtLvl: REAL;
	_bRecallManualLevel: BOOL;
	_fMinPctToBallast : REAL :=0.1;
END_VAR
VAR_OUTPUT
	fSP_Group	: REAL;
	bWriteValue : BOOL;
	bDimUp : BOOL;
	bDimDwn : BOOL;
	bOff : BOOL;
	bClMinCtrlVal: BOOL;
END_VAR
VAR_IN_OUT
	stPirSensorData		: ST_DALI_Sensor;
END_VAR
VAR
	fDiff: REAL;
	fDiffPct:REAL;
	fbStepTimer_TON: TON;
	fDiffAbs: REAL;
	bDoNothing: BOOL;
	bStep1: BOOL;
	bStep2: BOOL;
	bStep3: BOOL;
	bStep4: BOOL;
	bStep5: BOOL;
	bIncrease: BOOL;
	bDecrease: BOOL;
	fbStartUpVal: R_TRIG;
	fbStartUp: R_TRIG;
	fStepSize_1: REAL;
	fStepSize_2: REAL;
	fStepSize_3: REAL;
	fStepSize_4: REAL;
	fStepSize_5: REAL;
	fbTurnOff: R_TRIG;
	fbF_Trig: F_TRIG;
	fbBA_ValTrigf : FB_BA_ValTrigf;
	bTurnOff: BOOL;
	bWriteValueRTrig: BOOL;
	bActiveFB: BOOL;
	fbManFTRIG: F_TRIG;
	fHys: INT;
	fbRTrig_DataRead: R_TRIG;
	fbCheckOffValueDetect_TON: TON;
	fbTurnOffLight_TOF: TOF;
	fbBA_ValTrigLR : FB_BA_ValTrigF ;
	fbCheckCorrectLevel: TON;
	fbCheckReadBrightness: TON;
END_VAR

//New data from sensor
fbRTrig_DataRead(CLK:= stPirSensorData.bBrightnessRead);

//Checking the Read aren't keept high for long periode
fbCheckReadBrightness(IN:= stPirSensorData.bQueryBrightness , PT:= T#500MS , Q=> , ET=> );

IF fbCheckReadBrightness.Q THEN
	stPirSensorData.bQueryBrightness:= FALSE;
END_IF

(*Beregninger for differencen mellem SP og PV*)
IF fbRTrig_DataRead.Q THEN
	fDiff:=_fSP-_fPV;
	fDiffAbs:= ABS(_fSP-_fPV);
	IF fDiffAbs >0 THEN
		IF _fsp<= 0 THEN
			fDiffPct:= 100;
		ELSE
			fDiffPct:= (fDiffAbs / _fSP )*100;
		END_IF
	END_IF

	(*Check if we need to lower or raise the output *)
	bIncrease:= FALSE;
	bDecrease:= FALSE;

	IF fDiff < 0 THEN
		bDecrease:= TRUE;
	ELSE
		bIncrease:= TRUE;
	END_IF
END_IF


IF NOT _bTuningInProcess THEN

	IF NOT _bEnable THEN

		IF _bDimUp THEN
			IF _fActlLgtLvl = 0 THEN
				bClMinCtrlVal := TRUE;
			ELSE
				bClMinCtrlVal := FALSE;
				bDimUp:= TRUE;
			END_IF
		ELSE
				bClMinCtrlVal := FALSE;
				bDimUp:= FALSE;
		END_IF
		bDimDwn:= _bDimDown;


		IF _fSP > 0 THEN
			bActiveFB:= TRUE;
		ELSE
			bActiveFB:= FALSE;
		END_IF


	END_IF

	fbStartUpVal(CLK:=_bSyncVal, Q=> );

	IF (_fSP <> 0  AND _bEnable) OR fbStartUpVal.Q THEN
		fbTurnOff(CLK:= FALSE , Q=> );
		fbStepTimer_TON(IN:=_bEnable AND NOT fbStepTimer_TON.q , PT:=_tStepTime , Q=> , ET=> );
		IF fbStepTimer_TON.Q THEN
			stPirSensorData.bQueryBrightness := TRUE;
		END_IF

		(*Controlling the step rate*)

		bDoNothing:= FALSE;
		bStep1:= FALSE;
		bStep2:= FALSE;
		bStep3:= FALSE;
		bStep4:= FALSE;
		bStep5:= FALSE;

		IF _bStepModeCalculationOnSP THEN
			fStepSize_1:=_fSP *(_fSPStep1 / 100);
			fStepSize_2:=_fSP *(_fSPStep2 / 100);
			fStepSize_3:=_fSP *(_fSPStep3 / 100);
			fStepSize_4:=_fSP *(_fSPStep4 / 100);
			fStepSize_5:=_fSP *(_fSPStep5 / 100);
		ELSE
			fStepSize_1:=_fSPStep1;
			fStepSize_2:=_fSPStep2;
			fStepSize_3:=_fSPStep3;
			fStepSize_4:=_fSPStep4;
			fStepSize_5:=_fSPStep5;
		END_IF

		IF fDiffAbs <= _fStep1Limit THEN
			bDoNothing:= TRUE;
		END_IF

		IF (fDiffAbs > _fStep1Limit) AND  (fDiffAbs <= _fStep2Limit) THEN
			bStep1:= TRUE;
		END_IF

		IF (fDiffAbs > _fStep2Limit) AND  (fDiffAbs <= _fStep3Limit) THEN
			bStep2:= TRUE;
		END_IF

		IF (fDiffAbs > _fStep3Limit) AND  (fDiffAbs <= _fStep4Limit) THEN
			bStep3:= TRUE;
		END_IF

		IF (fDiffAbs > _fStep4Limit) AND  (fDiffAbs <= _fStep5Limit) THEN
			bStep4:= TRUE;
		END_IF

		IF (fDiffAbs > _fStep5Limit)  THEN
			bStep5:= TRUE;
		END_IF

	
//		IF (fbStepTimer_TON.Q) OR bTurnOff  THEN
		IF fbRTrig_DataRead.Q OR bTurnOff THEN
			stPirSensorData.bQueryBrightness:= FALSE;
			IF bStep1 THEN
				IF bDecrease THEN
				fSP_Group:=LIMIT (_fMinPctToBallast, (fSP_Group - fStepSize_1), 100);

				END_IF

				IF bIncrease THEN
					fSP_Group:=LIMIT (_fMinPctToBallast, (fSP_Group + fStepSize_1), 100);

				END_IF
			END_IF

			IF bStep2 THEN
				IF bDecrease THEN
					fSP_Group:=LIMIT (_fMinPctToBallast, (fSP_Group - fStepSize_2), 100);

				END_IF

				IF bIncrease THEN
					fSP_Group:=LIMIT (_fMinPctToBallast, (fSP_Group + fStepSize_2), 100);

				END_IF
			END_IF

			IF bStep3 THEN
				IF bDecrease THEN
					fSP_Group:=LIMIT (_fMinPctToBallast, (fSP_Group - fStepSize_3), 100);

				END_IF

				IF bIncrease THEN
					fSP_Group:=LIMIT (_fMinPctToBallast, (fSP_Group + fStepSize_3), 100);

				END_IF
			END_IF

			IF bStep4 THEN
				IF bDecrease THEN
					fSP_Group:=LIMIT (_fMinPctToBallast, (fSP_Group - fStepSize_4), 100);

				END_IF

				IF bIncrease THEN
					fSP_Group:=LIMIT (_fMinPctToBallast, (fSP_Group + fStepSize_4), 100);

				END_IF
			END_IF

			IF bStep5 THEN
				IF bDecrease THEN
					fSP_Group:=LIMIT (_fMinPctToBallast, (fSP_Group - fStepSize_5), 100);

				END_IF

				IF bIncrease THEN
					fSP_Group:=LIMIT (_fMinPctToBallast, (fSP_Group + fStepSize_5), 100);

		END_IF
			END_IF
		END_IF

		IF fbStartUpVal.Q THEN
			fSP_Group:= LIMIT(_fMinPctToBallast, (_fSyncVal),100);
		END_IF

		
	ELSE
		IF _fSP = 0 THEN
			fSP_Group:= 0;
		END_IF
	END_IF
ELSE
		fSP_Group:=_fSetValDct;
		bWriteValue:= _bSetValDct;
END_IF


IF _bRecallManualLevel THEN
		fSP_Group:=_fSetValDct;
		bWriteValue:= _bSetValDct;
END_IF

(*Lukker korrekt skrive bit, efter endt Tuning*)
	fbF_Trig(CLK:=_bTuningInProcess , Q=> );

	IF fbF_Trig.Q THEN
		bWriteValue:= FALSE;
	END_IF

fbTurnOffLight_TOF(IN:=((fSP_Group<> 0) ) , PT:= T#500MS );


fbCheckOffValueDetect_TON(IN:= (_bOff AND (_fActlLgtLvl > 0 )) AND NOT fbCheckOffValueDetect_TON.Q , PT:=T#500MS);

fbCheckCorrectLevel(IN:= (1 < ABS(_fActlLgtLvl- fSP_Group)) AND NOT fbCheckCorrectLevel.Q , PT:= T#500MS , Q=> , ET=> );

fbBA_ValTrigLR(
	bEn:=TRUE ,
	bRetrig:= fbTurnOff.Q OR fbCheckCorrectLevel.Q,
	fIn:=fSP_Group ,
	fHys:=0.5,
	fOut=> ,
	bSet=>);
	

fbManFTRIG(CLK:= bActiveFB, Q=> );

bWriteValue:= fbStartUpVal.Q OR fbBA_ValTrigLR.bSet OR fbManFTRIG.Q OR fbCheckOffValueDetect_TON.Q;

END_FUNCTION_BLOCK

// POUs/DALI/Power Control/FB_LightCtrl_1Group_OLD
FUNCTION_BLOCK FB_LightCtrl_1Group_OLD
VAR_INPUT
	_bEnable:BOOL;
	_bSyncVal:BOOL;
	_fSyncVal:REAL;
	_fSP : REAL;
	_fPV : REAL;
	_fStep1Limit: REAL;
	_fSPStep1 : REAL;
	_fStep2Limit: REAL;
	_fSPStep2 : REAL;
	_fStep3Limit: REAL;
	_fSPStep3 : REAL;
	_fStep4Limit: REAL;
	_fSPStep4 : REAL;
	_fStep5Limit: REAL;
	_fSPStep5 : REAL;
	_tStepTime : TIME;
	_bStepModeCalculationOnSP:BOOL;
	_bTuningInProcess: BOOL;
	_bSetValDct: BOOL;
	_fSetValDct: REAL;
	_bDimUp : BOOL;
	_bDimDown : BOOL;
	_bOff : BOOL;
	_fActlLgtLvl: REAL;
	_bRecallManualLevel: BOOL;
END_VAR
VAR_OUTPUT
	fSP_Group	: REAL;
	bWriteValue : BOOL;
	bDimUp : BOOL;
	bDimDwn : BOOL;
	bOff : BOOL;
	bClMinCtrlVal: BOOL;
END_VAR
VAR_IN_OUT
	stPirSensorData		: ST_DALI_Sensor;
END_VAR
VAR
	fDiff: REAL;
	fDiffPct:REAL;
	fbStepTimer_TON: TON;
	fDiffAbs: REAL;
	bDoNothing: BOOL;
	bStep1: BOOL;
	bStep2: BOOL;
	bStep3: BOOL;
	bStep4: BOOL;
	bStep5: BOOL;
	bIncrease: BOOL;
	bDecrease: BOOL;
	fbStartUpVal: R_TRIG;
	fbStartUp: R_TRIG;
	fStepSize_1: REAL;
	fStepSize_2: REAL;
	fStepSize_3: REAL;
	fStepSize_4: REAL;
	fStepSize_5: REAL;
	fbTurnOff: R_TRIG;
	fbF_Trig: F_TRIG;
	fbBA_ValTrigf : FB_BA_ValTrigf;
	bTurnOff: BOOL;
	bWriteValueRTrig: BOOL;
	bActiveFB: BOOL;
	fbManFTRIG: F_TRIG;
	fHys: INT;
END_VAR

(*Beregninger for differencen mellem SP og PV*)
	fDiff:=_fSP-_fPV;
	fDiffAbs:= ABS(_fSP-_fPV);
	IF fDiffAbs >0 THEN
		IF _fsp<= 0 THEN
			fDiffPct:= 100;
		ELSE
			fDiffPct:= (fDiffAbs / _fSP )*100;
		END_IF
	END_IF

	(*Check if we need to lower or raise the output *)
	bIncrease:= FALSE;
	bDecrease:= FALSE;


	IF fDiff < 0 THEN
		bDecrease:= TRUE;
	ELSE
		bIncrease:= TRUE;
	END_IF



IF NOT _bTuningInProcess THEN

	IF NOT _bEnable THEN
		IF _bDimUp THEN
			IF _fActlLgtLvl = 0 THEN
				bClMinCtrlVal := TRUE;
			ELSE
				bClMinCtrlVal := FALSE;
				bDimUp:= TRUE;
			END_IF
		ELSE
				bClMinCtrlVal := FALSE;
				bDimUp:= FALSE;
		END_IF
		bDimDwn:= _bDimDown;

		IF _fSP > 0 THEN
			bActiveFB:= TRUE;
		ELSE
			bActiveFB:= FALSE;
		END_IF


(*		fbTurnOff(CLK:=_bOff , Q=> );
		IF fbTurnOff.Q THEN
			fSP_Group:=0;
			fSP_Room:=0;
			fbDelaySendValueWrite(IN:=TRUE , PT:= (UDINT_TO_TIME(SystemTaskInfoArr[1].cycleTime)*2) , Q=> , ET=> );
			bWriteValueRTrig:= fbDelaySendValueWrite.Q
		END_IF
*)	END_IF

	IF _fSP <> 0  AND _bEnable  THEN
		fbTurnOff(CLK:= FALSE , Q=> );
		fbStepTimer_TON(IN:=_bEnable AND NOT fbStepTimer_TON.q , PT:=_tStepTime , Q=> , ET=> );
		fbStartUpVal(CLK:=_bSyncVal , Q=> );


		IF fbStartUpVal.Q THEN
			fSP_Group:=LIMIT(0, (_fSyncVal + fSP_Group), 100);
		END_IF


		(*Controlling the step rate*)

		bDoNothing:= FALSE;
		bStep1:= FALSE;
		bStep2:= FALSE;
		bStep3:= FALSE;
		bStep4:= FALSE;
		bStep5:= FALSE;

		IF _bStepModeCalculationOnSP THEN
			fStepSize_1:=_fSP * (_fSPStep1 / 100);
			fStepSize_2:=_fSP *( _fSPStep2 / 100);
			fStepSize_3:=_fSP *( _fSPStep3 / 100);
			fStepSize_4:=_fSP *( _fSPStep4 / 100);
			fStepSize_5:=_fSP *( _fSPStep5 / 100);
		ELSE
			fStepSize_1:=_fSPStep1;
			fStepSize_2:=_fSPStep2;
			fStepSize_3:= _fSPStep3;
			fStepSize_4:= _fSPStep4;
			fStepSize_5:=_fSPStep5;
		END_IF


		IF fDiffAbs <= _fStep1Limit THEN
			bDoNothing:= TRUE;
		END_IF

		IF (fDiffAbs > _fStep1Limit) AND  (fDiffAbs <= _fStep2Limit) THEN
			bStep1:= TRUE;
		END_IF

		IF (fDiffAbs > _fStep2Limit) AND  (fDiffAbs <= _fStep3Limit) THEN
			bStep2:= TRUE;
		END_IF

		IF (fDiffAbs > _fStep3Limit) AND  (fDiffAbs <= _fStep4Limit) THEN
			bStep3:= TRUE;
		END_IF

		IF (fDiffAbs > _fStep4Limit) AND  (fDiffAbs <= _fStep5Limit) THEN
			bStep4:= TRUE;
		END_IF

		IF (fDiffAbs > _fStep5Limit)  THEN
			bStep5:= TRUE;
		END_IF


		IF (fbStepTimer_TON.Q OR fbStartUp.Q) OR bTurnOff  THEN

			IF bStep1 THEN
				IF bDecrease THEN
					fSP_Group:=LIMIT (0, (fSP_Group - fStepSize_1), 100);
				END_IF

				IF bIncrease THEN
					fSP_Group:=LIMIT (0, (fSP_Group - fStepSize_1), 100);
				END_IF
			END_IF

			IF bStep2 THEN
				IF bDecrease THEN
					fSP_Group:=LIMIT (0, (fSP_Group - fStepSize_2), 100);
				END_IF

				IF bIncrease THEN
					fSP_Group:=LIMIT (0, (fSP_Group +  fStepSize_2),100);
				END_IF
			END_IF

			IF bStep3 THEN
				IF bDecrease THEN
					fSP_Group:=LIMIT (0, (fSP_Group - fStepSize_3), 100);
				END_IF

				IF bIncrease THEN
					fSP_Group:=LIMIT (0, (fSP_Group +  fStepSize_3),100);
				END_IF
			END_IF

			IF bStep4 THEN
				IF bDecrease THEN
					fSP_Group:=LIMIT (0, (fSP_Group - fStepSize_4), 100);
				END_IF

				IF bIncrease THEN
					fSP_Group:=LIMIT (0, (fSP_Group +  fStepSize_4),100);
				END_IF
			END_IF

			IF bStep5 THEN
				IF bDecrease THEN
					fSP_Group:=LIMIT (0, (fSP_Group - fStepSize_5), 100);
				END_IF

				IF bIncrease THEN
					fSP_Group:=LIMIT (0, (fSP_Group +  fStepSize_5),100);
		END_IF
			END_IF
		END_IF
	ELSE
		fSP_Group:= 0;

	END_IF
ELSE
		fSP_Group:=_fSetValDct;
		bWriteValue:= _bSetValDct;
END_IF


IF _bRecallManualLevel THEN
		fSP_Group:=_fSetValDct;
		bWriteValue:= _bSetValDct;
END_IF

(*Lukker korrekt skrive bit, efter endt Tuning*)
	fbF_Trig(CLK:=_bTuningInProcess , Q=> );

	IF fbF_Trig.Q THEN
		bWriteValue:= FALSE;
	END_IF

fbTurnOff(CLK:= _fSP = 0 , Q=> );

fbBA_ValTrigf(
	bEn:=TRUE ,
	bRetrig:= _bOff OR fbTurnOff.Q,
	fIn:=fSP_Group ,
	fHys:=0.5,
	fOut=> ,
	bSet=>bWriteValue);

fbManFTRIG(CLK:= bActiveFB, Q=> );

bWriteValue:= fbStartUpVal.Q OR fbBA_ValTrigf.bSet OR fbManFTRIG.Q;

END_FUNCTION_BLOCK

// POUs/DALI/Power Control/FB_LightCtrl_2Groups
FUNCTION_BLOCK FB_LightCtrl_2Groups
VAR_INPUT
	_bEnable:BOOL;
	_bSyncVal:BOOL;
	_fSyncVal:REAL;
	_fSP : REAL;
	_fPV : REAL;
	_fStep1Limit: REAL;
	_fSPStep1 : REAL;
	_fStep2Limit: REAL;
	_fSPStep2 : REAL;
	_fStep3Limit: REAL;
	_fSPStep3 : REAL;
	_fStep4Limit: REAL;
	_fSPStep4 : REAL;
	_fStep5Limit: REAL;
	_fSPStep5 : REAL;
	_tStepTime : TIME;
	_bStepModeCalculationOnSP:BOOL;
	_bTuningInProcess: BOOL;
	_bSetValDct: BOOL;
	_fSetValDct: REAL;
	_bDimUp : BOOL;
	_bDimDown : BOOL;
	_bOff : BOOL;
	_fRowOffset: REAL;
	_fActlLgtLvl_Prim: REAL;
	_fActlLgtLvl_Sec: REAL;
	_bRecallManualLevel: BOOL;
	_fMinOutputPowerLevel : REAL;
	_fMaxOutputPowerLevel : REAL;
	_DALI_LINE_NUM_SEC	: BYTE;
END_VAR
VAR_OUTPUT
	fSP_Window	: REAL;
	fSP_Room	: REAL;
	bWriteValue : BOOL;
	bDimUp : BOOL;
	bDimDwn : BOOL;
	bOff : BOOL;
	bClMinCtrlVal:BOOL;
END_VAR
VAR_IN_OUT
	stPirSensorData		: ST_DALI_Sensor;
END_VAR
VAR
	fDiff: REAL;
	fDiffPct:REAL;
	fbStepTimer_TON: TON;
	fDiffAbs: REAL;
	bDoNothing: BOOL;
	bStep1: BOOL;
	bStep2: BOOL;
	bStep3: BOOL;
	bStep4: BOOL;
	bStep5: BOOL;
	bIncrease: BOOL;
	bDecrease: BOOL;
	fbStartUpVal: R_TRIG;
	fbStartUp: R_TRIG;
	fStepSize_1: REAL;
	fStepSize_2: REAL;
	fStepSize_3: REAL;
	fStepSize_4: REAL;
	fStepSize_5: REAL;

	fbTurnOff: R_TRIG;
	fbF_Trig: F_TRIG;
	fbRTrig_DataRead: R_TRIG;

	fbBA_ValTrigf : FB_BA_ValTrigF;
	fbTurnOffAuto: R_TRIG;
	bTurnOff: BOOL;
	bWriteValueRTrig: BOOL;
	fbDelaysReleaseCtrl: TON;
	fbDelayResend_TON: TON;
	bReSendCmd: BOOL;
	fX0: REAL;
	fX1: REAL := 100;
	fY0: REAL;
	fY1: REAL := 100;
	fDeltaX: REAL;	
	fDeltaY: REAL;
	
	fSPWindowCalc: REAL;
	bEnableCtrl: BOOL;
	fbCheckReadBrightness: TON;
END_VAR

//New data from sensor
fbRTrig_DataRead(CLK:= stPirSensorData.bBrightnessRead);

//Checking the Read aren't keept high for long periode
fbCheckReadBrightness(IN:= stPirSensorData.bQueryBrightness , PT:= T#500MS , Q=> , ET=> );

IF fbCheckReadBrightness.Q OR fbRTrig_DataRead.Q THEN
	stPirSensorData.bQueryBrightness:= FALSE;
END_IF

fY0:=_fRowOffset*-1;
fDeltaY:= fY1-fY0;
fDeltaX :=fX1-fX0;
		
IF fDeltaX <=0 THEN			
	fDeltaX:=1;
END_IF


(*Beregninger for differencen mellem SP og PV*)
IF fbRTrig_DataRead.Q THEN
	fDiff:=_fSP-_fPV;
	fDiffAbs:= ABS(_fSP-_fPV);
	IF fDiffAbs >0 THEN
		IF _fsp<= 0 THEN
			fDiffPct:= 100;
		ELSE
			fDiffPct:= (fDiffAbs / _fSP )*100;
		END_IF
	END_IF

	(*Check if we need to lower or raise the output *)
	bIncrease:= FALSE;
	bDecrease:= FALSE;
	
	IF fDiff < 0 THEN
		bDecrease:= TRUE;
	ELSE
		bIncrease:= TRUE;
	END_IF
END_IF

//Continous calculating step size

bDoNothing:= FALSE;
bStep1:= FALSE;
bStep2:= FALSE;
bStep3:= FALSE;
bStep4:= FALSE;
bStep5:= FALSE;

IF _bStepModeCalculationOnSP THEN
	fStepSize_1:=_fSP * (_fSPStep1 / 100);
	fStepSize_2:=_fSP *( _fSPStep2 / 100);
	fStepSize_3:=_fSP *( _fSPStep3 / 100);
	fStepSize_4:=_fSP *( _fSPStep4 / 100);
	fStepSize_5:=_fSP *( _fSPStep5 / 100);
ELSE
	fStepSize_1:=_fSPStep1;
	fStepSize_2:=_fSPStep2;
	fStepSize_3:= _fSPStep3;
	fStepSize_4:= _fSPStep4;
	fStepSize_5:=_fSPStep5;
END_IF

IF fDiffPct <= _fStep1Limit THEN
	bDoNothing:= TRUE;
END_IF

IF (fDiffPct > _fStep1Limit) AND  (fDiffPct <= _fStep2Limit) THEN
	bStep1:= TRUE;
END_IF

IF (fDiffPct > _fStep2Limit) AND  (fDiffPct <= _fStep3Limit) THEN
	bStep2:= TRUE;
END_IF

IF (fDiffPct > _fStep3Limit) AND  (fDiffPct <= _fStep4Limit) THEN
	bStep3:= TRUE;
END_IF

IF (fDiffPct > _fStep4Limit) AND  (fDiffPct <= _fStep5Limit) THEN
	bStep4:= TRUE;
END_IF

IF (fDiffPct > _fStep5Limit)  THEN
	bStep5:= TRUE;
END_IF

//LightCtrlProcess
IF NOT _bTuningInProcess THEN
	IF NOT _bEnable THEN
		IF _bDimUp THEN
			IF _fActlLgtLvl_Prim = 0 OR (_fActlLgtLvl_Sec = 0 AND _DALI_LINE_NUM_SEC <> 0) THEN
				bClMinCtrlVal := TRUE;
			ELSE
				bClMinCtrlVal := FALSE;
				bDimUp:= TRUE;
			END_IF
		ELSE
				bClMinCtrlVal := FALSE;
				bDimUp:= FALSE;
		END_IF
		bDimDwn:= _bDimDown;

	END_IF

	IF _fSP <> 0  AND _bEnable  THEN
		fbTurnOff(CLK:= FALSE , Q=> );
		fbStepTimer_TON(IN:=_bEnable AND NOT fbStepTimer_TON.q , PT:=_tStepTime , Q=> , ET=> );
		
		fbDelaysReleaseCtrl(IN:= bEnableCtrl , PT:=T#5S , Q=> , ET=> );

		IF fbDelaysReleaseCtrl.Q THEN 

	 		IF fbStepTimer_TON.Q THEN
				stPirSensorData.bQueryBrightness := TRUE;
			END_IF

			(*Controlling the step rate*)
			IF (fbRTrig_DataRead.Q OR fbStartUp.Q) OR bTurnOff  THEN
				stPirSensorData.bQueryBrightness := FALSE;
				IF bStep1 THEN
					IF bDecrease THEN
						fSP_Room:=LIMIT (_fMinOutputPowerLevel, (fSP_Room - fStepSize_1), _fMaxOutputPowerLevel);
					END_IF
	
					IF bIncrease THEN
						fSP_Room:=LIMIT (_fMinOutputPowerLevel, (fSP_Room +  fStepSize_1), _fMaxOutputPowerLevel);
					END_IF
				END_IF
	
				IF bStep2 THEN
					IF bDecrease THEN
						fSP_Room:=LIMIT (_fMinOutputPowerLevel, (fSP_Room - fStepSize_2), _fMaxOutputPowerLevel);
					END_IF
	
					IF bIncrease THEN
						fSP_Room:=LIMIT (_fMinOutputPowerLevel, (fSP_Room +  fStepSize_2), _fMaxOutputPowerLevel);
					END_IF
				END_IF
	
				IF bStep3 THEN
					IF bDecrease THEN
						fSP_Room:=LIMIT (_fMinOutputPowerLevel, (fSP_Room - fStepSize_3), _fMaxOutputPowerLevel);
					END_IF
	
					IF bIncrease THEN
						fSP_Room:=LIMIT (_fMinOutputPowerLevel, (fSP_Room +  fStepSize_3), _fMaxOutputPowerLevel);
					END_IF
				END_IF
	
				IF bStep4 THEN
					IF bDecrease THEN
						fSP_Room:=LIMIT (_fMinOutputPowerLevel, (fSP_Room - fStepSize_4), _fMaxOutputPowerLevel);
					END_IF
	
					IF bIncrease THEN
						fSP_Room:=LIMIT (_fMinOutputPowerLevel, (fSP_Room +  fStepSize_4), _fMaxOutputPowerLevel);
					END_IF
				END_IF
	
				IF bStep5 THEN
					IF bDecrease THEN
						fSP_Room:=LIMIT (_fMinOutputPowerLevel, (fSP_Room - fStepSize_5), _fMaxOutputPowerLevel);
					END_IF
	
					IF bIncrease THEN
						fSP_Room:=LIMIT (_fMinOutputPowerLevel, (fSP_Room +  fStepSize_5), _fMaxOutputPowerLevel);
					END_IF
				END_IF
			END_IF
		END_IF
		
			fSPWindowCalc:= (fDeltaY / fDeltaX) * fSP_Room + fY0;
			fSP_Window:=LIMIT (0, (fSPWindowCalc),_fMaxOutputPowerLevel);
	ELSE
		fSP_Window:= 0;
		fSP_Room := 0;
	END_IF

	IF fbStartUpVal.Q THEN
		fSP_Room:= LIMIT(_fMinOutputPowerLevel,(_fSyncVal), _fMaxOutputPowerLevel);
	END_IF


ELSE
	fSP_Window:=_fSetValDct;
	fSP_Room:=_fSetValDct;
	bWriteValue:= _bSetValDct;
END_IF

fbStartUpVal(CLK:=_bSyncVal , Q=> );

IF fbStartUpVal.Q THEN
	fSP_Room:= LIMIT(_fMinOutputPowerLevel,(_fSyncVal), _fMaxOutputPowerLevel);
	fSPWindowCalc:= (fDeltaY / fDeltaX) * fSP_Room + fY0;
	fSP_Window:=LIMIT (0, (fSPWindowCalc),_fMaxOutputPowerLevel);
	bEnableCtrl:= TRUE;	
END_IF

IF _bRecallManualLevel THEN
	fSP_Window:=_fSetValDct;
	fSP_Room:=_fSetValDct;
	bWriteValue:= _bSetValDct;
END_IF

(*Lukker korrekt skrive bit, efter endt Tuning*)
fbF_Trig(CLK:=_bTuningInProcess , Q=> );

IF fbF_Trig.Q THEN
	bWriteValue:= FALSE;
END_IF

fbTurnOff(CLK:= _fSP = 0 , Q=> );

IF ((ABS(_fActlLgtLvl_Sec - fSP_Window) > 2) OR (ABS(_fActlLgtLvl_Prim - fSP_Room)> 2)) AND _bEnable THEN
	fbDelayResend_TON(IN:=TRUE , PT:= T#15S, Q=> , ET=> );
	IF fbDelayResend_TON.Q THEN
		bReSendCmd:= TRUE;
		fbDelayResend_TON(IN:=FALSE);
	ELSE
		bReSendCmd:= FALSE;
	END_IF
END_IF

fbBA_ValTrigf(
	bEn:=bEnableCtrl ,
	bRetrig:= _bOff OR fbTurnOff.Q OR bReSendCmd ,
	fIn:=(fSP_Room + fSP_Window) ,
	fHys:=0.5,
	fOut=> ,
	bSet=>bWriteValue);
	
IF _bOff OR fbTurnOff.Q AND NOT _bEnable THEN
	bEnableCtrl:= FALSE;
END_IF

END_FUNCTION_BLOCK

// POUs/DALI/Power Control/FB_LightCtrl_2Groups_Action
FUNCTION_BLOCK FB_LightCtrl_2Groups_Action
VAR_INPUT
	_bEnable:BOOL;
	_bSyncVal:BOOL;
	_fSyncVal:REAL;
	_fSP : REAL;
	_fPV : REAL;
	_fStep1Limit: REAL;
	_fSPStep1 : REAL;
	_fStep2Limit: REAL;
	_fSPStep2 : REAL;
	_fStep3Limit: REAL;
	_fSPStep3 : REAL;
	_fStep4Limit: REAL;
	_fSPStep4 : REAL;
	_fStep5Limit: REAL;
	_fSPStep5 : REAL;
	_tStepTime : TIME;
	_bStepModeCalculationOnSP:BOOL;
	_bTuningInProcess: BOOL;
	_bSetValDct: BOOL;
	_fSetValDct: REAL;
	_bDimUp : BOOL;
	_bDimDown : BOOL;
	_bOff : BOOL;
	_fRowOffset: REAL;
	_fActlLgtLvl_Prim: REAL;
	_fActlLgtLvl_Sec: REAL;
	_bRecallManualLevel: BOOL;
	_fMinOutputPowerLevel : REAL;
	_fMaxOutputPowerLevel : REAL;
END_VAR
VAR_OUTPUT
	fSP_Window	: REAL;
	fSP_Room	: REAL;
	bWriteValue : BOOL;
	bDimUp : BOOL;
	bDimDwn : BOOL;
	bOff : BOOL;
	bClMinCtrlVal:BOOL;
END_VAR
VAR_IN_OUT
	stPirSensorData		: ST_DALI_Sensor;
END_VAR
VAR
	fDiff: REAL;
	fDiffPct:REAL;
	fbStepTimer_TON: TON;
	fDiffAbs: REAL;
	bDoNothing: BOOL;
	bStep1: BOOL;
	bStep2: BOOL;
	bStep3: BOOL;
	bStep4: BOOL;
	bStep5: BOOL;
	bIncrease: BOOL;
	bDecrease: BOOL;
	fbStartUpVal: R_TRIG;
	fbStartUp: R_TRIG;
	fStepSize_1: REAL;
	fStepSize_2: REAL;
	fStepSize_3: REAL;
	fStepSize_4: REAL;
	fStepSize_5: REAL;

	fbTurnOff: R_TRIG;
	fbF_Trig: F_TRIG;
	fbRTrig_DataRead: R_TRIG;

	fbBA_ValTrigf : FB_BA_ValTrigF;
	fbTurnOffAuto: R_TRIG;
	bTurnOff: BOOL;
	bWriteValueRTrig: BOOL;
	fbDelaysReleaseCtrl: TON;
	fbDelayResend_TON: TON;
	bReSendCmd: BOOL;
	fX0: REAL;
	fX1: REAL := 100;
	fY0: REAL;
	fY1: REAL := 100;
	fDeltaX: REAL;	
	fDeltaY: REAL;
	
	fSPWindowCalc: REAL;
	bEnableCtrl: BOOL;
	fbCheckReadBrightness: TON;
END_VAR

//New data from sensor
fbRTrig_DataRead(CLK:= stPirSensorData.bBrightnessRead);

//Checking the Read aren't keept high for long periode
fbCheckReadBrightness(IN:= stPirSensorData.bQueryBrightness , PT:= T#500MS , Q=> , ET=> );

IF fbCheckReadBrightness.Q OR fbRTrig_DataRead.Q THEN
	stPirSensorData.bQueryBrightness:= FALSE;
END_IF

(*Beregninger for differencen mellem SP og PV*)
IF fbRTrig_DataRead.Q THEN
	fDiff:=_fSP-_fPV;
	fDiffAbs:= ABS(_fSP-_fPV);
	IF fDiffAbs >0 THEN
		IF _fsp<= 0 THEN
			fDiffPct:= 100;
		ELSE
			fDiffPct:= (fDiffAbs / _fSP )*100;
		END_IF
	END_IF

	(*Check if we need to lower or raise the output *)
	bIncrease:= FALSE;
	bDecrease:= FALSE;
	
	IF fDiff < 0 THEN
		bDecrease:= TRUE;
	ELSE
		bIncrease:= TRUE;
	END_IF
END_IF

//Continous calculating step size

bDoNothing:= FALSE;
bStep1:= FALSE;
bStep2:= FALSE;
bStep3:= FALSE;
bStep4:= FALSE;
bStep5:= FALSE;

IF _bStepModeCalculationOnSP THEN
	fStepSize_1:=_fSP * (_fSPStep1 / 100);
	fStepSize_2:=_fSP *( _fSPStep2 / 100);
	fStepSize_3:=_fSP *( _fSPStep3 / 100);
	fStepSize_4:=_fSP *( _fSPStep4 / 100);
	fStepSize_5:=_fSP *( _fSPStep5 / 100);
ELSE
	fStepSize_1:=_fSPStep1;
	fStepSize_2:=_fSPStep2;
	fStepSize_3:= _fSPStep3;
	fStepSize_4:= _fSPStep4;
	fStepSize_5:=_fSPStep5;
END_IF

IF fDiffPct <= _fStep1Limit THEN
	bDoNothing:= TRUE;
END_IF

IF (fDiffPct > _fStep1Limit) AND  (fDiffPct <= _fStep2Limit) THEN
	bStep1:= TRUE;
END_IF

IF (fDiffPct > _fStep2Limit) AND  (fDiffPct <= _fStep3Limit) THEN
	bStep2:= TRUE;
END_IF

IF (fDiffPct > _fStep3Limit) AND  (fDiffPct <= _fStep4Limit) THEN
	bStep3:= TRUE;
END_IF

IF (fDiffPct > _fStep4Limit) AND  (fDiffPct <= _fStep5Limit) THEN
	bStep4:= TRUE;
END_IF

IF (fDiffPct > _fStep5Limit)  THEN
	bStep5:= TRUE;
END_IF

//LightCtrlProcess
IF NOT _bTuningInProcess THEN
	IF _bEnable THEN
		A_Auto();	
	ELSE	
		A_Manuel();
	END_IF

	IF fbStartUpVal.Q THEN
		fSP_Room:= LIMIT(_fMinOutputPowerLevel,(_fSyncVal), _fMaxOutputPowerLevel);
	END_IF

		fY0:=_fRowOffset*-1;
		fDeltaY:= fY1-fY0;
		fDeltaX :=fX1-fX0;
				
		IF fDeltaX <=0 THEN			
			fDeltaX:=1;
		END_IF
ELSE
	
	A_Tuning();

END_IF

IF _bRecallManualLevel THEN
		fSP_Window:=_fSetValDct;
		fSP_Room:=_fSetValDct;
		bWriteValue:= _bSetValDct;
END_IF

(*Lukker korrekt skrive bit, efter endt Tuning*)
	fbF_Trig(CLK:=_bTuningInProcess , Q=> );

	IF fbF_Trig.Q THEN
		bWriteValue:= FALSE;
	END_IF


fbTurnOff(CLK:= _fSP = 0 , Q=> );

fbBA_ValTrigf(
	bEn:=TRUE ,
	bRetrig:= _bOff OR fbTurnOff.Q OR bReSendCmd,
	fIn:=(fSP_Room + fSP_Window) ,
	fHys:=0.5,
	fOut=> ,
	bSet=>bWriteValue);

ACTION A_Auto:
	IF _fSP <> 0  AND _bEnable  THEN
		fbTurnOff(CLK:= FALSE , Q=> );
		fbStepTimer_TON(IN:=_bEnable AND NOT fbStepTimer_TON.q , PT:=_tStepTime , Q=> , ET=> );
		fbStartUpVal(CLK:=_bSyncVal , Q=> );
		
		IF fbStartUpVal.Q THEN
			bEnableCtrl:= TRUE;
		END_IF
		
		fbDelaysReleaseCtrl(IN:= bEnableCtrl , PT:=T#5S , Q=> , ET=> );

		IF fbDelaysReleaseCtrl.Q THEN 

	 		IF fbStepTimer_TON.Q THEN
				stPirSensorData.bQueryBrightness := TRUE;
			END_IF

			(*Controlling the step rate*)
			IF (fbRTrig_DataRead.Q OR fbStartUp.Q) OR bTurnOff  THEN
				stPirSensorData.bQueryBrightness := FALSE;
				IF bStep1 THEN
					IF bDecrease THEN
						fSP_Room:=LIMIT (_fMinOutputPowerLevel, (fSP_Room - fStepSize_1), _fMaxOutputPowerLevel);
					END_IF
	
					IF bIncrease THEN
						fSP_Room:=LIMIT (_fMinOutputPowerLevel, (fSP_Room +  fStepSize_1), _fMaxOutputPowerLevel);
					END_IF
				END_IF
	
				IF bStep2 THEN
					IF bDecrease THEN
						fSP_Room:=LIMIT (_fMinOutputPowerLevel, (fSP_Room - fStepSize_2), _fMaxOutputPowerLevel);
					END_IF
	
					IF bIncrease THEN
						fSP_Room:=LIMIT (_fMinOutputPowerLevel, (fSP_Room +  fStepSize_2), _fMaxOutputPowerLevel);
					END_IF
				END_IF
	
				IF bStep3 THEN
					IF bDecrease THEN
						fSP_Room:=LIMIT (_fMinOutputPowerLevel, (fSP_Room - fStepSize_3), _fMaxOutputPowerLevel);
					END_IF
	
					IF bIncrease THEN
						fSP_Room:=LIMIT (_fMinOutputPowerLevel, (fSP_Room +  fStepSize_3), _fMaxOutputPowerLevel);
					END_IF
				END_IF
	
				IF bStep4 THEN
					IF bDecrease THEN
						fSP_Room:=LIMIT (_fMinOutputPowerLevel, (fSP_Room - fStepSize_4), _fMaxOutputPowerLevel);
					END_IF
	
					IF bIncrease THEN
						fSP_Room:=LIMIT (_fMinOutputPowerLevel, (fSP_Room +  fStepSize_4), _fMaxOutputPowerLevel);
					END_IF
				END_IF
	
				IF bStep5 THEN
					IF bDecrease THEN
						fSP_Room:=LIMIT (_fMinOutputPowerLevel, (fSP_Room - fStepSize_5), _fMaxOutputPowerLevel);
					END_IF
	
					IF bIncrease THEN
						fSP_Room:=LIMIT (_fMinOutputPowerLevel, (fSP_Room +  fStepSize_5), _fMaxOutputPowerLevel);
					END_IF
				END_IF
			END_IF
		END_IF
		
			fSPWindowCalc:= (fDeltaY / fDeltaX) * fSP_Room + fY0;
			fSP_Window:=LIMIT (0, (fSPWindowCalc),_fMaxOutputPowerLevel);
	ELSE
		fSP_Window:= 0;
		fSP_Room := 0;
	END_IF
	
	
	IF (ABS(_fActlLgtLvl_Sec - fSP_Window) > 2) OR (ABS(_fActlLgtLvl_Prim - fSP_Room)> 2) AND _bEnable THEN
		fbDelayResend_TON(IN:=TRUE , PT:= T#15S, Q=> , ET=> );
		IF fbDelayResend_TON.Q THEN
			bReSendCmd:= TRUE;
			fbDelayResend_TON(IN:=FALSE);
		ELSE
			bReSendCmd:= FALSE;
		END_IF
	END_IF
END_ACTION

ACTION A_Manuel:

		IF _bDimUp THEN
			IF _fActlLgtLvl_Prim = 0 OR _fActlLgtLvl_Sec = 0 THEN
				bClMinCtrlVal := TRUE;
			ELSE
				bClMinCtrlVal := FALSE;
				bDimUp:= TRUE;
			END_IF
		ELSE
				bClMinCtrlVal := FALSE;
				bDimUp:= FALSE;
		END_IF
		bDimDwn:= _bDimDown;
END_ACTION

ACTION A_Tuning:
	fSP_Window:=_fSetValDct;
	fSP_Room:=_fSetValDct;
	bWriteValue:= _bSetValDct;
END_ACTION

END_FUNCTION_BLOCK

// POUs/DALI/Power Control/FB_LightSwitch
FUNCTION_BLOCK FB_LightSwitch
VAR_INPUT
	bSwi			: BOOL;
	bSwiUp			: BOOL;
	bSwiDwn			: BOOL;
	udiSwiOvrTi		: UDINT;

	bUp				: BOOL;
	bDwn			: BOOL;

	bOn				: BOOL;
	bOff			: BOOL;

	eOnMod			: E_OnMode;
	fOnVal			: REAL;

	bClMinVal		: BOOL;
	bClMaxVal		: BOOL;
	bSetValDct		: BOOL;
	fSetValDct		: REAL;
	fActlLgtLvl 	: REAL;
END_VAR
VAR_OUTPUT
	stLgtCmd		: ST_LgtCmd;
END_VAR
VAR
	uiLgtCmdPulseTi	: UINT:=0;
	bInit			: BOOL;
	bLight			: BOOL;
	fbSwi			: FB_Click;
	fbSwiUp			: FB_Click;
	fbSwiDwn		: FB_Click;
	bToggleOn		: BOOL;
	bToggleOff		: BOOL;
	bDimDir			: BOOL;

	rtOff			: R_TRIG;
	rtClMinCtrlVal	: R_TRIG;
	rtClMaxCtrlVal	: R_TRIG;
	rtClOnVal		: R_TRIG;
	rtClRstVal		: R_TRIG;
	rtSetValDct		: R_TRIG;

	uiCmdStep		: USINT;
	tonCmdDurt		: TON;
	bOneCycle		: BOOL;

END_VAR

IF NOT bInit THEN
	bInit:=TRUE;
	bDimDir:=TRUE;
END_IF

(* + + + + + + + + + + + + + + + + + + + + + + + + + + + + + + + + + + + + + + + + + + + + *)
(*Beurteilung der angesteuerten Lichtaktoren über den Eingang lrActLgtLvl*)
bLight		:=(fActlLgtLvl<>0.0); (*Licht an/aus -> wichtig für toggle-Befehl*)

(* + + + + + + + + + + + + + + + + + + + + + + + + + + + + + + + + + + + + + + + + + + + + *)
(*Tastenfunktionen*)

fbSwi	(bSwitch:=bSwi,	tSwitchTime:=UDINT_TO_TIME(udiSwiOvrTi));
fbSwiUp	(bSwitch:=bSwiUp,	tSwitchTime:=UDINT_TO_TIME(udiSwiOvrTi));
fbSwiDwn(bSwitch:=bSwiDwn,	tSwitchTime:=UDINT_TO_TIME(udiSwiOvrTi));

bToggleOn	:= (fbSwi.bShortClick OR fbSwiUp.bShortClick OR fbSwiDwn.bShortClick) AND NOT bLight;
bToggleOff	:= (fbSwi.bShortClick OR fbSwiUp.bShortClick OR fbSwiDwn.bShortClick) AND bLight;

(* + + + + + + + + + + + + + + + + + + + + + + + + + + + + + + + + + + + + + + + + + + + + *)
(* Flankenbildung der Schaltbefehle *)
rtOff			(CLK:=(bOff AND (fActlLgtLvl>0)) OR bToggleOff);
rtClMinCtrlVal	(CLK:=((bOn OR bToggleOn) AND (eOnMod=e_ClMinVal)) OR bClMinVal);
rtClMaxCtrlVal	(CLK:=((bOn OR bToggleOn) AND (eOnMod=e_ClMaxVal)) OR bClMaxVal);
rtClOnVal		(CLK:=(bOn OR bToggleOn) AND (eOnMod=e_ClOnVal));
rtClRstVal		(CLK:=(bOn OR bToggleOn) AND (eOnMod=e_ClRstVal));
rtSetValDct		(CLK:=bSetValDct);

(* + + + + + + + + + + + + + + + + + + + + + + + + + + + + + + + + + + + + + + + + + + + + *)
(* Priorisierung aller Befehle und Schrittzuweisung *)
IF	(uiCmdStep=0)	THEN
	IF		fbSwi.bLongClick	AND (bDimDir OR NOT bLight)	THEN
				uiCmdStep:=10;
	ELSIF	fbSwi.bLongClick	AND NOT bDimDir 	THEN
				uiCmdStep:=20;
	ELSIF	fbSwiUp.bLongClick	THEN
				uiCmdStep:=13;
	ELSIF	fbSwiDwn.bLongClick	THEN
				uiCmdStep:=23;
	ELSIF	bUp		AND bLight	THEN
				uiCmdStep:=16;
	ELSIF	bDwn	AND bLight	THEN
				uiCmdStep:=26;


	ELSIF	rtOff.Q				THEN
				uiCmdStep:=30;
	ELSIF	rtClMinCtrlVal.Q	THEN
				uiCmdStep:=40;
	ELSIF	rtClMaxCtrlVal.Q	THEN
				uiCmdStep:=50;
	ELSIF	rtClOnVal.Q			THEN
				uiCmdStep:=60;
	ELSIF	rtClRstVal.Q		THEN
				uiCmdStep:=70;
	ELSIF	rtSetValDct.Q		THEN
				uiCmdStep:=80;
	END_IF
END_IF

(* + + + + + + + + + + + + + + + + + + + + + + + + + + + + + + + + + + + + + + + + + + + + *)
(*Kommandoausgabe*)
(*Dimmen = Dauerbefehl, Schalten = Kurz- bzw. Tastbefehl über Pulszeit*)

tonCmdDurt.PT:=UDINT_TO_TIME(uiLgtCmdPulseTi); (*Ausführungsdauer des Kommandos, da Trigger u.U. zu kurz*)

CASE uiCmdStep OF

0: (*Idle*);

10:(*fbSwi.bLongPress + bDimdir =TRUE -> Dauerbefehl*)
	IF NOT bLight		THEN
		stLgtCmd.bClMinCtrlVal := TRUE;
		stLgtCmd.bDimUp := FALSE;
	END_IF
	IF bLight		THEN
		stLgtCmd.bClMinCtrlVal := FALSE;
		stLgtCmd.bDimUp := TRUE;
	END_IF
	IF NOT fbSwi.bLongClick	THEN
		A_BA_LgtSwi_ResetCommands();
		bDimDir := FALSE;
		uiCmdStep:=0;
	END_IF

13:(*fbSwiUp.bLongPress -> Dauerbefehl*)
	IF NOT bLight		THEN
		stLgtCmd.bClMinCtrlVal := TRUE;
		stLgtCmd.bDimUp := FALSE;
	END_IF
	IF bLight		THEN
		stLgtCmd.bClMinCtrlVal := FALSE;
		stLgtCmd.bDimUp := TRUE;
	END_IF
	IF NOT fbSwiUp.bLongClick	THEN
		A_BA_LgtSwi_ResetCommands();
		bDimDir:=FALSE;
		uiCmdStep:=0;
	END_IF

16:(*bUp -> Dauerbefehl*)
	stLgtCmd.bDimUp	:= TRUE;
	IF NOT bUp	THEN
		A_BA_LgtSwi_ResetCommands();
		bDimDir := FALSE;
		uiCmdStep:=0;
	END_IF

20:(*fbSwi.bLongPress +bDimDir =FALSE-> Dauerbefehl*)
	stLgtCmd.bDimDwn := TRUE;
	IF NOT fbSwi.bLongClick	THEN
		A_BA_LgtSwi_ResetCommands();
		bDimDir:=TRUE;
		uiCmdStep:=0;
	END_IF

23:(*fbSwiDwn.bLongPress -> Dauerbefehl*)
	IF NOT bLight		THEN
		stLgtCmd.bClMaxCtrlVal := TRUE;
		stLgtCmd.bDimDwn := FALSE;
	END_IF
	IF bLight		THEN
		stLgtCmd.bClMinCtrlVal := FALSE;
		stLgtCmd.bDimDwn := TRUE;
	END_IF
	IF NOT fbSwiDwn.bLongClick	THEN
		A_BA_LgtSwi_ResetCommands();
		bDimDir := TRUE;
		uiCmdStep:=0;
	END_IF

26:(*bDwn -> Dauerbefehl*)
	stLgtCmd.bDimDwn := TRUE;
	IF NOT bDwn	THEN
		A_BA_LgtSwi_ResetCommands();
		bDimDir := TRUE;
		uiCmdStep:=0;
	END_IF

30:(*Off*)
	stLgtCmd.bOff:= TRUE;
	bDimDir := TRUE;
	A_BA_LgtSwi_WaitToReset();
40:(*Call MinCtrlVal*)
	stLgtCmd.bClMinCtrlVal := TRUE;
	bDimDir := TRUE;
	A_BA_LgtSwi_WaitToReset();
50:(*Call MaxCtrlVal*)
	stLgtCmd.bClMaxCtrlVal := TRUE;
	bDimDir := FALSE;
	A_BA_LgtSwi_WaitToReset();
60:(*Call OnValue*)
	stLgtCmd.bClOnVal := TRUE;
	stLgtCmd.lrOnVal:=fOnVal;
	A_BA_LgtSwi_WaitToReset();
70:(*Call ResetVal*)
	stLgtCmd.bClRstVal := TRUE;
	A_BA_LgtSwi_WaitToReset();
80:(*Call DirectValue*)
	stLgtCmd.bSetCtrlValDct := TRUE;
	stLgtCmd.fSetCtrlValDct:=fSetValDct;
	A_BA_LgtSwi_WaitToReset();
END_CASE

ACTION A_BA_LgtSwi_ResetCommands:
stLgtCmd.bOff			:= FALSE;
stLgtCmd.bClMinCtrlVal	:= FALSE;
stLgtCmd.bClMaxCtrlVal	:= FALSE;
stLgtCmd.bClOnVal		:= FALSE;
stLgtCmd.bClRstVal		:= FALSE;
stLgtCmd.bSetCtrlValDct	:= FALSE;
stLgtCmd.bDimUp			:= FALSE;
stLgtCmd.bDimDwn		:= FALSE;
stLgtCmd.bStpUp			:= FALSE;
stLgtCmd.bStpDwn		:= FALSE;
END_ACTION

ACTION A_BA_LgtSwi_WaitToReset:
tonCmdDurt(IN:=TRUE);
IF (uiLgtCmdPulseTi=0)	THEN
	IF bOneCycle	THEN
		A_BA_LgtSwi_ResetCommands();
		tonCmdDurt	(IN:=FALSE);
		bOneCycle	:=FALSE;
		uiCmdStep	:=0;
	ELSE
		bOneCycle :=TRUE;
	END_IF

ELSIF tonCmdDurt.Q	THEN
	A_BA_LgtSwi_ResetCommands();
	tonCmdDurt	(IN:=FALSE);
	bOneCycle	:=FALSE;
	uiCmdStep	:=0;
END_IF
END_ACTION

END_FUNCTION_BLOCK

// POUs/DALI/Power Control/FB_SearchStartUpLevel_EX
FUNCTION_BLOCK FB_SearchStartUpLevel_EX
VAR_INPUT
	bSearch				: BOOL;
	fSp					: REAL;
END_VAR
VAR_OUTPUT
	bSync				: BOOL;
	fSttUpCtrlVal		: REAL;
END_VAR
VAR
	nSearchStep 		:INT;
	fDeviation			: REAL;
	nSearch				: INT;
	fSp_Old				: REAL;
	bResearch			: BOOL;
	fbNewSearch 		: R_Trig;
END_VAR
VAR_IN_OUT
	stTuneData			: ST_TuneData_Ex;
	stPirSensorData		: ST_DALI_Sensor;
END_VAR

fDeviation:= fSp - stPirSensorData.fBrightness;

IF fSP <> fSp_Old THEN
	IF fDeviation < 0 THEN
		fSp_Old:= fSp;
		RETURN;
	ELSE
		bResearch:= TRUE;
	END_IF
END_IF

CASE nSearchStep OF

0: (*Waiting state*)
	fbNewSearch(CLK:= bSearch , Q=> );
	bSync:= FALSE;
	IF fbNewSearch.Q OR bResearch THEN
		nSearchStep:= 1;
		stPirSensorData.bQueryBrightness:= TRUE;
	END_IF

1:	
	IF stPirSensorData.bBrightnessRead THEN
		stPirSensorData.bQueryBrightness:= FALSE;
		nSearchStep:= 10;
		fSttUpCtrlVal := 0;
	END_IF
	
10:
	IF fDeviation<0 THEN
		fSttUpCtrlVal:=0;
	ELSE
		FOR nSearch:=0 TO 20 DO
			IF (stTuneData.arrLuxLevels[nSearch]>= fDeviation) THEN
				 IF (fDeviation <= stTuneData.arrLuxLevels[nSearch+1]) OR (nSearch=20)  THEN
					fSttUpCtrlVal:= nSearch*5;
					EXIT;
				END_IF
			ELSE
					fSttUpCtrlVal:=100;
			END_IF
		END_FOR
	END_IF

	nSearchStep:= 20;

20: 
	bSync:=TRUE;
	bResearch := FALSE;
	nSearch := 0;
	nSearchStep:= 0;
	fSp_Old:= fSp;

ELSE
	nSearchStep:= 0;
END_CASE

END_FUNCTION_BLOCK

// POUs/Folding_Doors/FB_ConnectRooms_3Pcs
FUNCTION_BLOCK FB_ConnectRooms_3Pcs
VAR_INPUT
	bConnectRooms 								: BOOL := FALSE;
	arrOnZone1_SepRoom						: ARRAY[1..nMaxNumOfRooms] OF BOOL;
	arrTopButtonZone1_SepRoom			: ARRAY[1..nMaxNumOfRooms] OF BOOL;
	arrBottomButtonZone1_SepRoom		: ARRAY[1..nMaxNumOfRooms] OF BOOL;
	//arrConnectedRooms						: ARRAY[1..nMaxNumOfRooms] OF BOOL;
END_VAR
VAR_IN_OUT
	arrstPirSensorData_SepRoom			: ARRAY[1..nMaxNumOfRooms] OF ST_DALI_Sensor;
	arrstPirSensorData_ConnRoom			: ARRAY[1..nMaxNumOfRooms] OF ST_DALI_Sensor;
END_VAR

VAR_OUTPUT
	arrTopButtonZone1_ConnRoom			: ARRAY[1..nMaxNumOfRooms] OF BOOL;
	arrBottomButtonZone1_ConnRoom	: ARRAY[1..nMaxNumOfRooms] OF BOOL;
	arrOverride_ConnRoom						: ARRAY[1..nMaxNumOfRooms] OF BOOL := [nMaxNumOfRooms(FALSE)];
END_VAR
VAR
	fbOverrideRTrig								: Tc2_Standard.R_TRIG;
	//nRoomId												: UINT;
END_VAR
VAR CONSTANT
	nMaxNumOfRooms							: UINT := 3;												//<--- CHANGE MAX NUMBER OF ROOMS HERE
END_VAR


A_ButtonLogic();
A_OverrideLogic();
A_SensorLogic();

ACTION A_ButtonLogic:
IF bConnectRooms THEN
	arrTopButtonZone1_ConnRoom[1] := arrTopButtonZone1_SepRoom[1] OR arrTopButtonZone1_SepRoom[2] OR arrTopButtonZone1_SepRoom[3];
	arrTopButtonZone1_ConnRoom[2] := arrTopButtonZone1_ConnRoom[1];
	arrTopButtonZone1_ConnRoom[3] := arrTopButtonZone1_ConnRoom[1];
	arrBottomButtonZone1_ConnRoom[1] := arrBottomButtonZone1_SepRoom[1] OR arrBottomButtonZone1_SepRoom[2] OR arrBottomButtonZone1_SepRoom[3];
	arrBottomButtonZone1_ConnRoom[2] := arrBottomButtonZone1_ConnRoom[1];
	arrBottomButtonZone1_ConnRoom[3] := arrBottomButtonZone1_ConnRoom[1];
ELSE
	arrTopButtonZone1_ConnRoom := arrTopButtonZone1_SepRoom;
	arrBottomButtonZone1_ConnRoom := arrBottomButtonZone1_SepRoom;
END_IF
END_ACTION

ACTION A_OverrideLogic:
fbOverrideRTrig(CLK := bConnectRooms);
IF (arrOnZone1_SepRoom[1] OR arrOnZone1_SepRoom[2] OR arrOnZone1_SepRoom[3]) AND fbOverrideRTrig.Q THEN
	arrOverride_ConnRoom[1] :=TRUE;
	arrOverride_ConnRoom[2] :=TRUE;
	arrOverride_ConnRoom[3] :=TRUE;
ELSE
	arrOverride_ConnRoom[1] := FALSE;
	arrOverride_ConnRoom[2] := FALSE;
	arrOverride_ConnRoom[3] := FALSE;
END_IF
END_ACTION

ACTION A_SensorLogic:
IF bConnectRooms THEN
	//Input fra sensorer samles
	arrstPirSensorData_ConnRoom[1].fBrightness			:= MIN(arrstPirSensorData_SepRoom[1].fBrightness, arrstPirSensorData_SepRoom[2].fBrightness, arrstPirSensorData_SepRoom[3].fBrightness);
	arrstPirSensorData_ConnRoom[1].bPrc						:= arrstPirSensorData_SepRoom[1].bPrc OR arrstPirSensorData_SepRoom[2].bPrc OR arrstPirSensorData_SepRoom[3].bPrc;
	arrstPirSensorData_ConnRoom[1].bBrightnessRead	:= arrstPirSensorData_SepRoom[1].bBrightnessRead OR arrstPirSensorData_SepRoom[2].bBrightnessRead OR arrstPirSensorData_SepRoom[3].bBrightnessRead;
	arrstPirSensorData_ConnRoom[2].fBrightness			:= arrstPirSensorData_ConnRoom[1].fBrightness;
	arrstPirSensorData_ConnRoom[2].bPrc					:= arrstPirSensorData_ConnRoom[1].bPrc;
	arrstPirSensorData_ConnRoom[2].bBrightnessRead	:= arrstPirSensorData_ConnRoom[1].bBrightnessRead;
	arrstPirSensorData_ConnRoom[3].fBrightness			:= arrstPirSensorData_ConnRoom[1].fBrightness;
	arrstPirSensorData_ConnRoom[3].bPrc					:= arrstPirSensorData_ConnRoom[1].bPrc;
	arrstPirSensorData_ConnRoom[3].bBrightnessRead	:= arrstPirSensorData_ConnRoom[1].bBrightnessRead;

	//Output til sensorer fordeles
	IF arrstPirSensorData_ConnRoom[1].bQueryBrightness OR arrstPirSensorData_ConnRoom[2].bQueryBrightness OR arrstPirSensorData_ConnRoom[3].bQueryBrightness THEN
		arrstPirSensorData_SepRoom[1].bQueryBrightness := TRUE;
		arrstPirSensorData_SepRoom[2].bQueryBrightness := TRUE;
		arrstPirSensorData_SepRoom[3].bQueryBrightness := TRUE;
	ELSE
		arrstPirSensorData_SepRoom[1].bQueryBrightness := FALSE;
		arrstPirSensorData_SepRoom[2].bQueryBrightness := FALSE;
		arrstPirSensorData_SepRoom[3].bQueryBrightness := FALSE;
	END_IF
ELSE
	//Input fra sensorer samles uden ændring
	arrstPirSensorData_ConnRoom[1].fBrightness			:= arrstPirSensorData_SepRoom[1].fBrightness;
	arrstPirSensorData_ConnRoom[1].bPrc						:= arrstPirSensorData_SepRoom[1].bPrc;
	arrstPirSensorData_ConnRoom[1].bBrightnessRead	:= arrstPirSensorData_SepRoom[1].bBrightnessRead;
	arrstPirSensorData_ConnRoom[2].fBrightness			:= arrstPirSensorData_SepRoom[2].fBrightness;
	arrstPirSensorData_ConnRoom[2].bPrc						:= arrstPirSensorData_SepRoom[2].bPrc;
	arrstPirSensorData_ConnRoom[2].bBrightnessRead 	:= arrstPirSensorData_SepRoom[2].bBrightnessRead;
	arrstPirSensorData_ConnRoom[3].fBrightness			:= arrstPirSensorData_SepRoom[3].fBrightness;
	arrstPirSensorData_ConnRoom[3].bPrc						:= arrstPirSensorData_SepRoom[3].bPrc;
	arrstPirSensorData_ConnRoom[3].bBrightnessRead	:= arrstPirSensorData_SepRoom[3].bBrightnessRead;
	
	//Output til sensorer fordeles uden ændring
	IF arrstPirSensorData_ConnRoom[1].bQueryBrightness THEN
		arrstPirSensorData_SepRoom[1].bQueryBrightness := TRUE;
	ELSE
		arrstPirSensorData_SepRoom[1].bQueryBrightness := FALSE;
	END_IF
	IF arrstPirSensorData_ConnRoom[2].bQueryBrightness THEN
		arrstPirSensorData_SepRoom[2].bQueryBrightness := TRUE;
	ELSE
		arrstPirSensorData_SepRoom[2].bQueryBrightness := FALSE;
	END_IF
	IF arrstPirSensorData_ConnRoom[3].bQueryBrightness THEN
		arrstPirSensorData_SepRoom[3].bQueryBrightness := TRUE;
	ELSE
		arrstPirSensorData_SepRoom[3].bQueryBrightness := FALSE;
	END_IF
END_IF
END_ACTION

END_FUNCTION_BLOCK

// POUs/Folding_Doors/FB_ConnectRooms_xPcs
FUNCTION_BLOCK FB_ConnectRooms_xPcs
VAR_INPUT
	bConnectRooms								: BOOL;
	arrOnZone1_SepRoom						: ARRAY[1..nMaxNumOfRooms] OF BOOL;
	arrTopButtonZone1_SepRoom			: ARRAY[1..nMaxNumOfRooms] OF BOOL;
	arrBottomButtonZone1_SepRoom		: ARRAY[1..nMaxNumOfRooms] OF BOOL;
	arrConnRooms									: ARRAY[1..nMaxNumOfRooms] OF BOOL;
END_VAR
VAR_IN_OUT
	arrstPirSensorData_SepRoom				: ARRAY[1..nMaxNumOfRooms] OF ST_DALI_Sensor;
	arrstPirSensorData_ConnRoom			: ARRAY[1..nMaxNumOfRooms] OF ST_DALI_Sensor;
END_VAR

VAR_OUTPUT
	arrTopButtonZone1_ConnRoom			: ARRAY[1..nMaxNumOfRooms] OF BOOL;
	arrBottomButtonZone1_ConnRoom		: ARRAY[1..nMaxNumOfRooms] OF BOOL;
	arrOverride_ConnRoom						: ARRAY[1..nMaxNumOfRooms] OF BOOL := [nMaxNumOfRooms(FALSE)];
END_VAR
VAR
	fbOverrideRTrig								: Tc2_Standard.R_TRIG;
	nRoomId											: UINT;
	OnZone1Tmp									: BOOL := FALSE;
	bTopButtonTmp								: BOOL := FALSE;
	bBottomButtonTmp							: BOOL := FALSE;
	bOverrideTmp									: BOOL := FALSE;
	fBrightnessTmp									: REAL := 1023;
	bPrcTmp											: BOOL := FALSE;
	bBrightnessReadTmp							: BOOL := FALSE;
	bQueryBrightnessTmp						: BOOL := FALSE;
END_VAR
VAR CONSTANT
	nMaxNumOfRooms								: UINT := DALI_Param.byMaxNumOfFoldingDoors+1;
END_VAR

A_ButtonLogic();
A_OverrideLogic();
A_SensorLogic();

ACTION A_ButtonLogic:

IF bConnectRooms THEN
	bTopButtonTmp := FALSE;
	bBottomButtonTmp := FALSE;
	FOR nRoomId := 1 TO nMaxNumOfRooms DO
		IF arrConnRooms[nRoomId] THEN
			bTopButtonTmp := bTopButtonTmp OR arrTopButtonZone1_SepRoom[nRoomId];
			bBottomButtonTmp := bBottomButtonTmp OR arrBottomButtonZone1_SepRoom[nRoomId];
		END_IF
	END_FOR
	FOR nRoomId := 1 TO nMaxNumOfRooms DO
		IF arrConnRooms[nRoomId] THEN
			arrTopButtonZone1_ConnRoom[nRoomId] := bTopButtonTmp;
			arrBottomButtonZone1_ConnRoom[nRoomId] := bBottomButtonTmp;
		ELSE
			arrTopButtonZone1_ConnRoom[nRoomId] := arrTopButtonZone1_SepRoom[nRoomId];
			arrBottomButtonZone1_ConnRoom[nRoomId] := arrBottomButtonZone1_SepRoom[nRoomId];
		END_IF
	END_FOR
END_IF
END_ACTION

ACTION A_OverrideLogic:

fbOverrideRTrig(CLK := bConnectRooms);
FOR nRoomId := 1 TO nMaxNumOfRooms DO
		IF arrConnRooms[nRoomId] THEN
			bOverrideTmp := bOverrideTmp OR arrOnZone1_SepRoom[nRoomId];
		END_IF
	END_FOR
	
IF bOverrideTmp AND fbOverrideRTrig.Q THEN
	FOR nRoomId := 1 TO nMaxNumOfRooms DO
		IF arrConnRooms[nRoomId] THEN
			arrOverride_ConnRoom[nRoomId] := TRUE;
		ELSE
			arrOverride_ConnRoom[nRoomId] := FALSE;
		END_IF
	END_FOR
ELSE
	FOR nRoomId := 1 TO nMaxNumOfRooms DO
			arrOverride_ConnRoom[nRoomId] := FALSE;
	END_FOR
END_IF
(*
	FOR nRoomId := 1 TO nMaxNumOfRooms DO
		IF NOT arrConnRooms[nRoomId] THEN
			arrOverride_ConnRoom[nRoomId] := FALSE;
		END_IF
	END_FOR
END_IF
*)
END_ACTION

ACTION A_SensorLogic:

IF bConnectRooms THEN
	//Input fra sensorer samles
	fBrightnessTmp := 1023;
	bPrcTmp := FALSE;
	bBrightnessReadTmp := FALSE;
	FOR nRoomId := 1 TO nMaxNumOfRooms DO
		IF arrConnRooms[nRoomId] THEN
			fBrightnessTmp := MIN(fBrightnessTmp, arrstPirSensorData_SepRoom[nRoomId].fBrightness);
			bPrcTmp := bPrcTmp OR arrstPirSensorData_SepRoom[nRoomId].bPrc;
			bBrightnessReadTmp := bBrightnessReadTmp OR arrstPirSensorData_SepRoom[nRoomId].bBrightnessRead;
		END_IF
	END_FOR
	FOR nRoomId := 1 TO nMaxNumOfRooms DO
		IF arrConnRooms[nRoomId] THEN
			arrstPirSensorData_ConnRoom[nRoomId].fBrightness := fBrightnessTmp;
			arrstPirSensorData_ConnRoom[nRoomId].bPrc := bPrcTmp;
			arrstPirSensorData_ConnRoom[nRoomId].bBrightnessRead := bBrightnessReadTmp;
		END_IF
	END_FOR

	//Output til sensorer fordeles
	bQueryBrightnessTmp := FALSE;
	FOR nRoomId := 1 TO nMaxNumOfRooms DO
		IF arrConnRooms[nRoomId] THEN
			bQueryBrightnessTmp := bQueryBrightnessTmp OR arrstPirSensorData_ConnRoom[nRoomId].bQueryBrightness;
		END_IF
	END_FOR
	FOR nRoomId := 1 TO nMaxNumOfRooms DO
		IF arrConnRooms[nRoomId] THEN
			IF bQueryBrightnessTmp THEN
				arrstPirSensorData_SepRoom[nRoomId].bQueryBrightness := TRUE;
			ELSE
				arrstPirSensorData_SepRoom[nRoomId].bQueryBrightness := FALSE;
			END_IF
		END_IF
	END_FOR
	
	FOR nRoomId := 1 TO nMaxNumOfRooms DO
		IF NOT arrConnRooms[nRoomId] THEN
			arrstPirSensorData_ConnRoom[nRoomId].fBrightness			:= arrstPirSensorData_SepRoom[nRoomId].fBrightness;
			arrstPirSensorData_ConnRoom[nRoomId].bPrc						:= arrstPirSensorData_SepRoom[nRoomId].bPrc;
			arrstPirSensorData_ConnRoom[nRoomId].bBrightnessRead	:= arrstPirSensorData_SepRoom[nRoomId].bBrightnessRead;
			IF arrstPirSensorData_ConnRoom[nRoomId].bQueryBrightness THEN
				arrstPirSensorData_SepRoom[nRoomId].bQueryBrightness := TRUE;
			ELSE
				arrstPirSensorData_SepRoom[nRoomId].bQueryBrightness := FALSE;
			END_IF
		END_IF
	END_FOR
END_IF
END_ACTION

END_FUNCTION_BLOCK

// POUs/Folding_Doors/FB_FoldingDoor
FUNCTION_BLOCK FB_FoldingDoor
VAR_INPUT
	bFoldingDoorOpen 						: BOOL;
	arrOnZone1									: ARRAY[1..2] OF BOOL;
	arrTopButtonZone1						: ARRAY[1..2] OF BOOL;
	arrBottomButtonZone1					: ARRAY[1..2] OF BOOL;
END_VAR
VAR_IN_OUT
	arrstPirSensorData						: ARRAY[1..2] OF ST_DALI_Sensor;
	arrstPirSensorDataComb				: ARRAY[1..2] OF ST_DALI_Sensor;
END_VAR

VAR_OUTPUT
	arrTopButtonZone1Comb				: ARRAY[1..2] OF BOOL;
	arrBottomButtonZone1Comb			: ARRAY[1..2] OF BOOL;
	bOverride										: BOOL := FALSE;
END_VAR
VAR
	fbOverrideRTrig							: Tc2_Standard.R_TRIG;
END_VAR

A_ButtonLogic();
A_OverrideLogic();
A_SensorLogic();

ACTION A_ButtonLogic:
IF bFoldingDoorOpen THEN
	arrTopButtonZone1Comb[1] := arrTopButtonZone1[1] OR arrTopButtonZone1[2];
	arrTopButtonZone1Comb[2] := arrTopButtonZone1Comb[1];
	arrBottomButtonZone1Comb[1] := arrBottomButtonZone1[1] OR arrBottomButtonZone1[2];
	arrBottomButtonZone1Comb[2] := arrBottomButtonZone1Comb[1];
ELSE
	arrTopButtonZone1Comb := arrTopButtonZone1;
	arrBottomButtonZone1Comb := arrBottomButtonZone1;
END_IF
END_ACTION

ACTION A_OverrideLogic:
fbOverrideRTrig(CLK := bFoldingDoorOpen);
IF (arrOnZone1[1] OR arrOnZone1[2]) AND fbOverrideRTrig.Q THEN
	bOverride := TRUE;
ELSE
	bOverride := FALSE;
END_IF
END_ACTION

ACTION A_SensorLogic:
IF bFoldingDoorOpen THEN
	//Input fra sensorer samles
	arrstPirSensorDataComb[1].fBrightness			:= MIN(arrstPirSensorData[1].fBrightness, arrstPirSensorData[2].fBrightness);
	arrstPirSensorDataComb[1].bPrc					:= arrstPirSensorData[1].bPrc OR arrstPirSensorData[2].bPrc;
	arrstPirSensorDataComb[1].bBrightnessRead	:= arrstPirSensorData[1].bBrightnessRead OR arrstPirSensorData[2].bBrightnessRead;
	arrstPirSensorDataComb[2].fBrightness			:= arrstPirSensorDataComb[1].fBrightness;
	arrstPirSensorDataComb[2].bPrc					:= arrstPirSensorDataComb[1].bPrc;
	arrstPirSensorDataComb[2].bBrightnessRead	:= arrstPirSensorDataComb[1].bBrightnessRead;

	//Output til sensorer fordeles
	IF arrstPirSensorDataComb[1].bQueryBrightness OR arrstPirSensorDataComb[2].bQueryBrightness THEN
		arrstPirSensorData[1].bQueryBrightness := TRUE;
		arrstPirSensorData[2].bQueryBrightness := TRUE;
	ELSE
		arrstPirSensorData[1].bQueryBrightness := FALSE;
		arrstPirSensorData[2].bQueryBrightness := FALSE;
	END_IF
ELSE
	//Input fra sensorer samles uden ændring
	arrstPirSensorDataComb[1].fBrightness			:= arrstPirSensorData[1].fBrightness;
	arrstPirSensorDataComb[1].bPrc					:= arrstPirSensorData[1].bPrc;
	arrstPirSensorDataComb[1].bBrightnessRead	:= arrstPirSensorData[1].bBrightnessRead;
	arrstPirSensorDataComb[2].fBrightness			:= arrstPirSensorData[2].fBrightness;
	arrstPirSensorDataComb[2].bPrc					:= arrstPirSensorData[2].bPrc;
	arrstPirSensorDataComb[2].bBrightnessRead := arrstPirSensorData[2].bBrightnessRead;
	
	//Output til sensorer fordeles uden ændring
	IF arrstPirSensorDataComb[1].bQueryBrightness THEN
		arrstPirSensorData[1].bQueryBrightness := TRUE;
	ELSE
		arrstPirSensorData[1].bQueryBrightness := FALSE;
	END_IF
	IF arrstPirSensorDataComb[2].bQueryBrightness THEN
		arrstPirSensorData[2].bQueryBrightness := TRUE;
	ELSE
		arrstPirSensorData[2].bQueryBrightness := FALSE;
	END_IF
END_IF
END_ACTION

END_FUNCTION_BLOCK

// POUs/Folding_Doors/FB_FoldingDoorCtrl_2Pcs
FUNCTION_BLOCK FB_FoldingDoorCtrl_2Pcs
VAR_INPUT
	arrFoldingDoorOpen 							: ARRAY[1..DALI_Param.byMaxNumOfFoldingDoors] OF BOOL;
	bFoldingDoorOpenTmp					: BOOL;
	
	arrRoomName									: ARRAY[1..nMaxNumOfRooms] OF STRING(12) := [(nMaxNumOfRooms)('NoName')];
	arrOnZone1_SepRoom						: ARRAY[1..nMaxNumOfRooms] OF BOOL;
	arrTopButtonZone1_SepRoom			: ARRAY[1..nMaxNumOfRooms] OF BOOL;
	arrBottomButtonZone1_SepRoom		: ARRAY[1..nMaxNumOfRooms] OF BOOL;
END_VAR
VAR_IN_OUT
	arrstPirSensorData_SepRoom				: ARRAY[1..nMaxNumOfRooms] OF ST_DALI_Sensor;
	arrstPirSensorData_ConnRoom			: ARRAY[1..nMaxNumOfRooms] OF ST_DALI_Sensor;
END_VAR

VAR_OUTPUT
	arrTopButtonZone1_ConnRoom				: ARRAY[1..nMaxNumOfRooms] OF BOOL;
	arrBottomButtonZone1_ConnRoom			: ARRAY[1..nMaxNumOfRooms] OF BOOL;
	arrOverride_ConnRoom							: ARRAY[1..nMaxNumOfRooms] OF BOOL := [(nMaxNumOfRooms)(FALSE)];
END_VAR
VAR
	fbOverrideRTrig							: Tc2_Standard.R_TRIG;
	nConfigId										: UINT;
	nStateId										: UINT;
	byFoldingDoorId							: BYTE;
	
	arrfbConnectRooms						: ARRAY[0..nNumOfConfigs-1] OF FB_ConnectRooms_xPcs; //Will be more instances than neccessary for nNumOfFoldingDoors > 2, but 
	
END_VAR
VAR CONSTANT
	nMaxNumOfRooms				: BYTE := DALI_Param.byMaxNumOfFoldingDoors+1;
	byNumOfFoldingDoors			: BYTE := 2;																																									//<--- CHANGE NUMBER OF FOLDING DOORS < nMaxNumOfFoldingDoors HERE
	
	//Number of possible configurations is ALWAYS 2 to the power of the number of folding doors	
	nNumOfConfigs					: UINT := TO_UINT(EXPT(2, byNumOfFoldingDoors));
	
	//Initializing possible configurations for arrFoldingDoorOpen with zero-indexing, where byNumOfFoldingDoors = 2
	arrConfigList									: ARRAY[0..nNumOfConfigs-1] OF ARRAY[1..byNumOfFoldingDoors] OF BOOL := [										//<--- CHANGE CONFIGURATION INITIALIZATION
																																			[FALSE,FALSE],
																																			[TRUE,FALSE],
																																			[FALSE,TRUE],
																																			[TRUE,TRUE]	];
																																	
	arrConnRooms								: ARRAY[0..nNumOfConfigs-1] OF ARRAY[1..nMaxNumOfRooms] OF BOOL := [
																																			[FALSE, FALSE, FALSE],		//Which rooms to connect in state 0
																																			[TRUE, TRUE, FALSE],		//Which rooms to connect in state 1
																																			[FALSE, TRUE, TRUE],		//Which rooms to connect in state 2
																																			[TRUE, TRUE, TRUE]		];	//Which rooms to connect in state 3
END_VAR

//Config Selector
FOR nConfigId := 0 TO (nNumOfConfigs-1) DO
	bFoldingDoorOpenTmp := TRUE;
	FOR byFoldingDoorId := 1 TO DALI_Param.byMaxNumOfFoldingDoors DO
		bFoldingDoorOpenTmp := bFoldingDoorOpenTmp AND (arrFoldingDoorOpen[byFoldingDoorId] = arrConfigList[nConfigId][byFoldingDoorId]); 
	END_FOR
	IF bFoldingDoorOpenTmp THEN
		nStateId := nConfigId;
		arrfbConnectRooms[nConfigId].bConnectRooms := TRUE;
	ELSE
		arrfbConnectRooms[nConfigId].bConnectRooms := FALSE;
	END_IF
END_FOR

CASE nStateId OF
	0: 	A_State0(); //No Change
	
	1: A_State1(); //An instance of connecting two rooms
	
	2:  A_State2(); //An instance of connecting two rooms
	
	3: A_State3(); //Instance of connecting three rooms
END_CASE

ACTION A_State0:

arrfbConnectRooms[0](
	arrOnZone1_SepRoom := arrOnZone1_SepRoom,
	arrTopButtonZone1_SepRoom := arrTopButtonZone1_SepRoom,
	arrBottomButtonZone1_SepRoom := arrBottomButtonZone1_SepRoom,
	arrConnRooms := arrConnRooms[0],
	arrstPirSensorData_SepRoom := arrstPirSensorData_SepRoom,
	arrstPirSensorData_ConnRoom := arrstPirSensorData_ConnRoom,
	arrTopButtonZone1_ConnRoom => arrTopButtonZone1_ConnRoom,
	arrBottomButtonZone1_ConnRoom => arrBottomButtonZone1_ConnRoom,
	arrOverride_ConnRoom => arrOverride_ConnRoom);
END_ACTION

ACTION A_State1:

arrfbConnectRooms[1](
	arrOnZone1_SepRoom := arrOnZone1_SepRoom,
	arrTopButtonZone1_SepRoom := arrTopButtonZone1_SepRoom,
	arrBottomButtonZone1_SepRoom := arrBottomButtonZone1_SepRoom,
	arrConnRooms := arrConnRooms[1],
	arrstPirSensorData_SepRoom := arrstPirSensorData_SepRoom,
	arrstPirSensorData_ConnRoom := arrstPirSensorData_ConnRoom,
	arrTopButtonZone1_ConnRoom => arrTopButtonZone1_ConnRoom,
	arrBottomButtonZone1_ConnRoom => arrBottomButtonZone1_ConnRoom,
	arrOverride_ConnRoom => arrOverride_ConnRoom);
END_ACTION

ACTION A_State2:

arrfbConnectRooms[2](
	arrOnZone1_SepRoom := arrOnZone1_SepRoom,
	arrTopButtonZone1_SepRoom := arrTopButtonZone1_SepRoom,
	arrBottomButtonZone1_SepRoom := arrBottomButtonZone1_SepRoom,
	arrConnRooms := arrConnRooms[2],
	arrstPirSensorData_SepRoom := arrstPirSensorData_SepRoom,
	arrstPirSensorData_ConnRoom := arrstPirSensorData_ConnRoom,
	arrTopButtonZone1_ConnRoom => arrTopButtonZone1_ConnRoom,
	arrBottomButtonZone1_ConnRoom => arrBottomButtonZone1_ConnRoom,
	arrOverride_ConnRoom => arrOverride_ConnRoom);
END_ACTION

ACTION A_State3:

arrfbConnectRooms[3](
	arrOnZone1_SepRoom := arrOnZone1_SepRoom,
	arrTopButtonZone1_SepRoom := arrTopButtonZone1_SepRoom,
	arrBottomButtonZone1_SepRoom := arrBottomButtonZone1_SepRoom,
	arrConnRooms := arrConnRooms[3],
	arrstPirSensorData_SepRoom := arrstPirSensorData_SepRoom,
	arrstPirSensorData_ConnRoom := arrstPirSensorData_ConnRoom,
	arrTopButtonZone1_ConnRoom => arrTopButtonZone1_ConnRoom,
	arrBottomButtonZone1_ConnRoom => arrBottomButtonZone1_ConnRoom,
	arrOverride_ConnRoom => arrOverride_ConnRoom);
END_ACTION

END_FUNCTION_BLOCK

// POUs/Internals/FB_FunctionType_A
(*
Lys tænder eller slukker ved betjening af tryk.
Lys dæmper ned til fLuxDim lux efter tPIRDim-tid (init 15min) uden aktivitet og slukkes efter tPIROff-tid (init 30min).

TRYKFUNKTIONER:
	Trykfunktion for knap til DALI-lys (med eller uden pendler).
		Tangent top:
			- Kort tryk - tænder/slukker
			- Langt tryk - varieres lys-niveauet op
		Tangent bund:
			- Kort tryk - tænder/slukker lys
			- Langt tryk - varieres lys-niveauet ned
		Hvis lys tændes med et kort tryk, sættes lokale i auto
		Hvis lys slukkes med kort tryk, sættes lokale i manuel
		Hvis et langt tryk aktiveres, sættes lokalet i manuel
		
	Trykfunktion for særskilt knap til PENDLER.
		Tangent top:
			- Kort tryk- tænd/sluk pendler
		Tangent bund:
			- Kort tryk - tænd/sluk pendler
		
	Trykfunktion for knap til OVERSTYRING:
		Tangent top:
			- Kort tryk - tænder DALI-lys og pendler og sætter lokale i auto
		Tangent bund:
			- Kort tryk - slukker DALI-lys og pendler og sætter lokale i manuel
		
PIR-FUNKTION:
	Ved tændt DALI-lys og ingen aktivitet i lokalet efter :
		15min (indstilleligt): DALI-Lys dæmpes til 200 lux (indstilleligt)
		30min (indstilleligt): DALI-lys og pendler slukker

	Ved slukket DALI-lys og ingen aktivitet i lokalet efter :
		15min (indstilleligt): Ingen ændring
		30min (indstilleligt): pendler slukker, hvis de er tændte og lokalet sættes i auto
		
	Ved slukket lys og lokale i auto og aktivitet:
		DALI-lys tænder
		Pendler tænder, hvis der ikke findes en særskilt knap
		
ZONER:
	Zone 1: Loftarmaturer Rum og Vindue
	Zone 2: Supplerende belysning (evt pendler)
*)

FUNCTION_BLOCK FB_FunctionType_A
VAR_INPUT
	bTopButtonZone1 			: BOOL;
	bBottomButtonZone1		: BOOL;
	bButtonZone2 				: BOOL;
	bNoButtons						: BOOL	:= FALSE;
	bTopButtonOverride		: BOOL	:= FALSE;
	bBottomButtonOverride	: BOOL	:= FALSE;
	bPIR 								: BOOL	:=TRUE;
	fLuxOn 							: REAL	:= 500;
	fLuxDim 							: REAL	:= 200;
	tPIRDim 							: TIME	:= T#15M;
	tPIROff 							: TIME	:= T#30M;
END_VAR
VAR_OUTPUT
	fLuxZone1 				: REAL;
	bDimUp					: BOOL:= FALSE;
	bDimDwn 				: BOOL:= FALSE;
	bOnZone1 				: BOOL;
	bOffZone1 				: BOOL:= TRUE;
	bAutoZone1 				: BOOL:= TRUE;
	
	bAutoZone2 				: BOOL:= TRUE;
	bOnZone2 				: BOOL;
	bOffZone2 				: BOOL:= TRUE;
	
END_VAR
VAR
	fbShortLongPressTopZone1 		:	FB_Click;
	fbShortLongPressBottomZone1	:	FB_Click;
	fbShortLongPresZone2 				:	FB_Click;
	fbShortLongPressTopOverride	:	FB_Click;
	fbShortLongPressBottomOverride	: FB_Click;

	fbTofDim, fbTofOff 		: TOF;
	fbFtrigDim, fbFtrigOff 	: F_TRIG;
	fbRTrig_DimUp 				: R_TRIG;
	fbRTrig_DimDwn			: R_TRIG;
	bDimUpActive					: BOOL;
	bDimDownActive			: BOOL;
END_VAR
VAR CONSTANT
	tShortClick 			: TIME :=T#250MS;
END_VAR

//Selecting function for override button
(* short click TOP *)
fbShortLongPressTopOverride(bSwitch:= bTopButtonOverride, tSwitchTime:= tShortClick);
IF fbShortLongPressTopOverride.bShortClick THEN		(* SHORT click *)
	bDimDownActive := FALSE;
	bDimUpActive := FALSE;
	fLuxZone1:= fLuxOn;
	bAutoZone1 := TRUE;
	bOnZone1:= TRUE;
	bOffZone1:= FALSE;
	bOnZone2 := TRUE;
	bOffZone2 := FALSE;
	bAutoZone2 := TRUE;
END_IF

(* short click Bottom *)
fbShortLongPressBottomOverride(bSwitch:= bBottomButtonOverride, tSwitchTime:= tShortClick);
IF fbShortLongPressBottomOverride.bShortClick THEN		(* SHORT click *)
	bDimDownActive := FALSE;
	bDimUpActive := FALSE;
	fLuxZone1:= 0;
	bAutoZone1 := FALSE;
	bOnZone1:= FALSE;
	bOffZone1:= TRUE;
	bOnZone2:= FALSE;
	bOffZone2:= TRUE;
	bAutoZone2:=FALSE;
END_IF


//Selecting function for Zone 1 Buttons
(* short click TOP*)
fbShortLongPressTopZone1(bSwitch := bTopButtonZone1, tSwitchTime := tShortClick);
IF fbShortLongPressTopZone1.bShortClick THEN		(* SHORT click *)
	bDimDownActive := FALSE;
	bDimUpActive := FALSE;
	IF NOT bOnZone1 THEN
		fLuxZone1:= fLuxOn;
		bAutoZone1 := TRUE;
		bOnZone1:= TRUE;
		bOffZone1:= FALSE;
	ELSE
		fLuxZone1:= 0;
		bAutoZone1 := FALSE;
		bOnZone1:= FALSE;
		bOffZone1:= TRUE;
	END_IF
END_IF

//Dim up activation
fbRTrig_DimUp(CLK:=(fbShortLongPressTopZone1.bLongClick));// OR fbShortLongPressTopOverride.bLongClick));
IF fbRTrig_DimUp.Q AND NOT (fbShortLongPressBottomZone1.bShortClick OR fbShortLongPressBottomOverride.bShortClick) THEN
	bDimUpActive:= TRUE;
	bDimDownActive := FALSE;
ELSE
	bDimUpActive := FALSE;
END_IF

//long click TOP
IF bTopButtonZone1 THEN // OR bTopButtonOverride THEN
	IF fbShortLongPressTopZone1.bLongClick THEN // OR fbShortLongPressTopOverride.bLongClick THEN
		fLuxZone1 := fLuxOn;
		bAutoZone1 := FALSE;
		bOnZone1:= TRUE;
		bOffZone1:= FALSE;
		IF bDimUpActive THEN
			bDimUp:= TRUE;
		ELSE
			bDimUp:= FALSE;
		END_IF
	END_IF
ELSE
	bDimUp	:= FALSE;
END_IF

(* short click BOTTOM*)
fbShortLongPressBottomZone1(bSwitch := bBottomButtonZone1, tSwitchTime := tShortClick);
IF fbShortLongPressBottomZone1.bShortClick THEN		(* SHORT click *)
	bDimDownActive := FALSE;
	bDimUpActive :=FALSE;
	IF	 bOnZone1 THEN
		fLuxZone1:= 0;
		bAutoZone1 := FALSE;
		bOnZone1:= FALSE;
		bOffZone1:= TRUE;
	ELSE
		fLuxZone1:= fLuxOn;
		bAutoZone1 := TRUE;
		bOnZone1:= TRUE;
		bOffZone1:= FALSE;
	END_IF
END_IF

//Dim down activation
fbRTrig_DimDwn(CLK:=(fbShortLongPressBottomZone1.bLongClick)); // OR fbShortLongPressBottomOverride.bLongClick));
IF fbRTrig_DimDwn.Q AND NOT (fbShortLongPressTopZone1.bShortClick OR fbShortLongPressTopOverride.bShortClick) THEN
	bDimDownActive:= TRUE;
	bDimUpActive := FALSE;
ELSE
	bDimDownActive := FALSE;
END_IF

// Long click BOTTOM
IF bBottomButtonZone1 THEN // OR bBottomButtonOverride THEN
	IF fbShortLongPressBottomZone1.bLongClick THEN // OR fbShortLongPressBottomOverride.bLongClick THEN
		fLuxZone1 := fLuxOn;
		bAutoZone1 := FALSE;
		bOnZone1:= TRUE;
		bOffZone1:= FALSE;
		IF bDimDownActive THEN
			bDimDwn:= TRUE;
		ELSE
			bDimDwn:= FALSE;
		END_IF
	END_IF
ELSE
	bDimDwn	:= FALSE;
END_IF

//Selecting function for Zone 2 Buttons
(* short click *)
fbShortLongPresZone2(bSwitch := bButtonZone2, tSwitchTime := tShortClick);
IF fbShortLongPresZone2.bShortClick THEN		(* SHORT click *)
	IF bOnZone2 THEN
		bAutoZone2 := TRUE;
		bOnZone2:= FALSE;
		bOffZone2:= TRUE;			
	ELSE
		bAutoZone2 := TRUE;
		bOnZone2:= TRUE;
		bOffZone2:= FALSE;		
	END_IF
END_IF

(* PIR function for automatic*)
	//Set the Lux ON SP to output if the room is in DIM mode and a person re-enter the room.
	IF bAutoZone1 AND bPIR AND bOnZone1 AND (fLuxZone1 = fLuxDim) THEN
		fLuxZone1:= fLuxOn;
	END_IF
	//Set the lux ON SP to output if a person enters AND the room is off AND room is auto
	IF bPIR AND bOffZone1 AND bAutoZone1 THEN
		bOnZone1	:=	TRUE;
		bOffZone1	:= FALSE;
		fLuxZone1	:= fLuxOn;
		IF bNoButtons THEN
			bOnZone2		:= TRUE;
			bOffZone2		:= FALSE;
			bAutoZone2	:= TRUE;
		END_IF
	END_IF
	
	//PIR delay time to dim
	fbTofDim(IN := (	fbShortLongPressTopZone1.bShortClick OR fbShortLongPressBottomZone1.bShortClick OR
								fbShortLongPressTopZone1.bLongClick OR fbShortLongPressBottomZone1.bLongClick) OR
								fbShortLongPressTopOverride.bShortClick OR fbShortLongPressBottomOverride.bShortClick OR
								bPIR, PT := tPIRDim);
	fbFtrigDim(CLK := fbTofDim.Q);
	
	//PIR delay time to off
	fbTofOff(IN := (	fbShortLongPressTopZone1.bShortClick OR fbShortLongPressBottomZone1.bShortClick OR
								fbShortLongPressTopZone1.bLongClick OR fbShortLongPressBottomZone1.bLongClick) OR
								fbShortLongPressTopOverride.bShortClick OR fbShortLongPressBottomOverride.bShortClick OR
								bPIR, PT := tPIROff);
	fbFtrigOff(CLK := fbTofOff.Q);
	
	IF fbFtrigDim.Q AND bOnZone1 THEN (* DIM light*)
			IF (fLuxZone1 > fLuxDim) THEN
				fLuxZone1:= fLuxDim;
				bOnZone1:= TRUE;
				bOffZone1:= FALSE;
			END_IF
	END_IF

	IF fbFtrigOff.Q THEN					(* Light Off *)
		bOnZone1		:= FALSE;
		bOffZone1		:= TRUE;
		bAutoZone1	:=TRUE;
		fLuxZone1		:= 0;
		bOnZone2		:= FALSE;
		bOffZone2		:= TRUE;
		bAutoZone2	:= TRUE;
	END_IF

//This makes sure that a new setpoint for fLuxOn is activated immediately
IF bAutoZone1 AND bOnZone1 AND fLuxZone1<>fLuxDim AND NOT fbShortLongPressBottomOverride.bShortClick THEN
	fLuxZone1 := fLuxOn;
END_IF

END_FUNCTION_BLOCK

// POUs/Misc/FB_ClockPulse
FUNCTION_BLOCK FB_ClockPulse
VAR_INPUT
	bGenerateClockPulses	: BOOL;
	tTimeInterval			: TIME;
	tPulseTime				: TIME;
END_VAR
VAR_OUTPUT
	bPulse	: BOOL;
END_VAR
VAR
	tonInterval		: TON;
	tp				: TP;						
	
END_VAR

IF bGenerateClockPulses THEN
	tonInterval(IN:= NOT (tonInterval.Q OR tp.Q), PT:= tTimeInterval);
	tp(IN:= tonInterval.Q, PT:= tPulseTime);
	bPulse := tp.Q;
END_IF

END_FUNCTION_BLOCK

// POUs/Misc/FB_CountOnHours
FUNCTION_BLOCK FB_CountOnHours
(*
The FB takes as in_out an UINT and adds 1 when an hour has passed on a rising edge if both bEnableHourCount is TRUE and bPauseCount is FALSE for the duration.
If bEnableHourCount is true a and bPauseCount is also true, the time reached before the pause is stored and reinstated as PV when bPauseCount is true on a rising edge
The in_out can be stored as persistent and the FB will use the stored value as after a download or restart.
The reached time - 0< tTimePaused< 1h -  before adding 1 to the output will be lost during download or restart.
An overflow precaution is implemented, which can be stored as persistent
*)
VAR_INPUT
	bEnableHourCount		: BOOL := TRUE;
	bPauseCount				: BOOL;
END_VAR
VAR_IN_OUT
	uiOnHours				: UINT;
	byOverflowCount			: BYTE;
END_VAR
VAR
	tPT						: TIME := T#60m;
	fbPause					: R_TRIG;
	tonHour					: TON;
	tTimePaused				: TIME;
	bHourPulse				: BOOL;
	fbRTrig_HourPulse		: R_TRIG;
	uiMaxOnHours			: UINT := 65535;
	bMaxReached				: BOOL;
	fbRTrig_MaxReached		: R_TRIG;
END_VAR

//Reset the PT
IF NOT bEnableHourCount OR tonHour.Q THEN
tTimePaused := T#0s;
END_IF

//Detect the Pause
fbPause(CLK := bPauseCount);

//Keep the Time
IF fbPause.Q THEN
tTimePaused := tTimePaused + tonHour.ET;
END_IF

//TON
tonHour(
IN	:= bEnableHourCount AND NOT (bPauseCount OR tonHour.Q),
PT	:= (tPT - tTimePaused),
Q	=> bHourPulse
);

//Count hours
fbRTrig_HourPulse(CLK:= bHourPulse);
IF fbRTrig_HourPulse.Q THEN
uiOnHours:= uiOnHours + 1;			//This makes sure the output can be stored as a persistent variable.
END_IF

//Resets uiOnHours when max is reached, which is 65535 OnHours ~ 7.5 OnYears, and counts up byOverflowCount by one
IF uiOnHours = uiMaxOnHours THEN
	bMaxReached:= TRUE;
ELSE
	bMaxReached:= FALSE;
END_IF

fbRTrig_MaxReached(CLK:= bMaxReached);
IF fbRTrig_MaxReached.Q THEN
	uiMaxOnHours:= 0;
	byOverflowCount:= byOverflowCount + 1;	
END_IF

END_FUNCTION_BLOCK

// POUs/Misc/FB_TwoVal_SelectOne_RTrigChange
FUNCTION_BLOCK FB_TwoVal_SelectOne_RTrigChange
VAR_INPUT
	bEnableSelection		: BOOL := TRUE;
	bEnableOverride		: BOOL := FALSE;
	nOverRideValue		: UINT := 30;
	nMaxValOut				: UINT;
END_VAR
VAR_IN_OUT
	nValIn1					: UINT;
	nValIn2					: UINT;
END_VAR
VAR_OUTPUT
	nValOut					: UINT;
END_VAR
VAR
	bValIn1Changed			: BOOL;// := FALSE;
	bValIn2Changed			: BOOL;// := FALSE;
	fbRTrig_ValIn1Change	: R_TRIG;
	fbRTrig_ValIn2Change	: R_TRIG;
	bRTrig_ValIn1Change		: BOOL;
	bRTrig_ValIn2Change		: BOOL;	
	
	nSelStepId				: UINT := 0;
END_VAR

{region "Enable"}
IF bEnableSelection AND nMaxValOut>0 THEN
{region "Value 1 changed"}
	IF nValIn1>nMaxValOut THEN
		nValIn1	:= nMaxValOut;
	END_IF

	IF (nValIn1<>nValOut) THEN
		bValIn1Changed	:= TRUE;	
	ELSE
		bValIn1Changed	:= FALSE;
	END_IF

	fbRTrig_ValIn1Change(CLK:=bValIn1Changed, Q=> bRTrig_ValIn1Change);
	IF bRTrig_ValIn1Change THEN
		nValIn2		:= nValIn1;
		nValOut		:= nValIn1;
	END_IF	
{endregion}
{region "Value 2 changed"}
	IF nValIn2>nMaxValOut THEN
		nValIn2	:= nMaxValOut;
	END_IF

	IF (nValIn2<>nValOut) THEN
		bValIn2Changed	:= TRUE;	
	ELSE
		bValIn2Changed	:= FALSE;
	END_IF

	fbRTrig_ValIn2Change(CLK:=bValIn2Changed, Q=> bRTrig_ValIn2Change);
	IF bRTrig_ValIn2Change AND NOT bValIn1Changed THEN
		nValIn1		:= nValIn2;
		nValOut		:= nValIn2;
	END_IF
{endregion}
{region "Override value"}
	IF bEnableOverride THEN
		nValOut := nOverRideValue;
		nValIn1 := nOverRideValue;
		nValIn2 := nOverRideValue;
	END_IF	
{endregion}
ELSE
	nValOut		:= 0;	
END_IF

END_FUNCTION_BLOCK

// POUs/Modbus/FB_ReadAHPirData
FUNCTION_BLOCK FB_ReadAHPirData
VAR_INPUT
	bReadAHPirData				: BOOL;
	sIPAddr						: STRING(15);
	nMBAddr						: WORD;
END_VAR
VAR_IN_OUT
	nMBDataBuffer				: UINT;
END_VAR
VAR_OUTPUT
	arrAH_NeighborRoomsPir		: ARRAY[0..15] OF BOOL;
END_VAR
VAR
	fbMBReadRegs				: FB_MBReadRegs;
END_VAR

fbMBReadRegs(	sIPAddr		:= sIPAddr,
				nTCPPort	:= 502,
				nUnitID		:= 255,
				nQuantity	:= SIZEOF(nMBDataBuffer)/2,
				nMBAddr		:= nMBAddr,
				cbLength	:= SIZEOF(nMBDataBuffer),
				pDestAddr	:= ADR(nMBDataBuffer),
				bExecute	:= bReadAHPirData,
				tTimeout	:= T#2S
			);

arrAH_NeighborRoomsPir[0] := nMBDataBuffer.0;
arrAH_NeighborRoomsPir[1] := nMBDataBuffer.1;
arrAH_NeighborRoomsPir[2] := nMBDataBuffer.2;
arrAH_NeighborRoomsPir[3] := nMBDataBuffer.3;
arrAH_NeighborRoomsPir[4] := nMBDataBuffer.4;
arrAH_NeighborRoomsPir[5] := nMBDataBuffer.5;
arrAH_NeighborRoomsPir[6] := nMBDataBuffer.6;
arrAH_NeighborRoomsPir[7] := nMBDataBuffer.7;
arrAH_NeighborRoomsPir[8] := nMBDataBuffer.8;
arrAH_NeighborRoomsPir[9] := nMBDataBuffer.9;
arrAH_NeighborRoomsPir[10] := nMBDataBuffer.10;
arrAH_NeighborRoomsPir[11] := nMBDataBuffer.11;
arrAH_NeighborRoomsPir[12] := nMBDataBuffer.12;
arrAH_NeighborRoomsPir[13] := nMBDataBuffer.13;
arrAH_NeighborRoomsPir[14] := nMBDataBuffer.14;
arrAH_NeighborRoomsPir[15] := nMBDataBuffer.15;

END_FUNCTION_BLOCK

// POUs/Scheduling/FB_TODScheduling
FUNCTION_BLOCK FB_TODScheduling
VAR_INPUT
	arrTODSchedule					: ARRAY[1..4] OF TOD;
	tdMidnight						: TOD := TOD#0:0:0;
	tdMorning						: TOD := TOD#6:0:0;
	tdMidDay						: TOD := TOD#12:0:0;
	tdEvening						: TOD := TOD#18:0:0;
	
	tCheckDuration					: TIME:= T#5S;
END_VAR
VAR_OUTPUT
	bStartTask						: BOOL;
END_VAR
VAR
	stLocalSystemTime 		: TIMESTRUCT;
	fbLocalSystemTime 		: FB_LocalSystemTime;
	bGetTime 				: BOOL := TRUE;
	tTimeOut 				: TIME := DEFAULT_ADS_TIMEOUT;
	bLocalSystemTimeValid	: BOOL;
	tzID       				: E_TimeZoneID := eTimeZoneID_Invalid;
	
	tdSystemTime			: TOD;
	
	byTODIdx				: BYTE;
END_VAR

fbLocalSystemTime(
	sNetID:= '', 
	bEnable:= bGetTime, 
	dwCycle:= 2, // cycle time (in seconds) , Synchronization  every 2 seconds.
	dwOpt:= 1, //Bit 0: If this is set, the Windows system time is additionally synchronized cyclically with the hardware clock (RTC) (corresponds to the function NT_SetTimeToRTCTime).
	tTimeout:= tTimeOut, 
	bValid=> bLocalSystemTimeValid, 
	systemTime=> stLocalSystemTime, 
	tzID=> tzID);
	
tdSystemTime := SYSTEMTIME_TO_TOD(systemTime := stLocalSystemTime);

FOR byTODIdx := 1 TO 4 DO
	IF	tdSystemTime > arrTODSchedule[byTODIdx] AND tdSystemTime < (arrTODSchedule[byTODIdx] + tCheckDuration) THEN
		bStartTask:= TRUE;
	ELSE
		bStartTask := FALSE;
	END_IF
END_FOR

END_FUNCTION_BLOCK

// POUs/Templates/FB_Light_Type_A
FUNCTION_BLOCK FB_Light_Type_A
VAR_INPUT	
	nZoneID						: UDINT;
	bButtonZone1				: BOOL;
	bBottomButtonZone1			: BOOL;
	bButtonZone2				: BOOL;
	bTopButtonOverride		: BOOL;
	bBottomButtonOverride	: BOOL;
	bNoButtons					: BOOL;
	fLuxOn 						: REAL;
	fLuxDim						: REAL;
	tPIRDim						: TIME;
	tPIROff						: TIME;
	fOffsetSec					: REAL;
	bReInit						: BOOL;
	stDaliSetup					: ST_DALI_RoomSetup;
	ipCommunication_Prim		: I_DALICommunication;
	ipCommunication_Sec			: I_DALICommunication;
	ipCommunication_Supl		: I_DALICommunication;
	fMinOutputPowerLevelRoom 	: REAL;
	fMaxOutputPowerLevelRoom	: REAL;
	nCycleTimeInMS				: UDINT;
	bRunTuning 					: BOOL;
END_VAR
VAR_OUTPUT
	bOccupiedRoom 	: BOOL;
	bError_Prim 	: BOOL;
	nError_Prim 	: UINT;
END_VAR
VAR
	fbBallast					: FB_Light_Ballast;
	fbLightCtrl					: FB_FunctionType_A ;
	fbShortLongPresZone1 		: FB_Click;
	fbShortLongPressBottomZone1 : FB_Click;
	fbShortLongPresZone2 		: FB_Click;

	stLgtCmd_Prim				: ST_LgtCmd;
	stLgtCmd_Sec				: ST_LgtCmd;
	stLgtCmd_Supl				: ST_LgtCmd;
	
	fbLightCtrl_2Rows			: FB_LightCtrl_2Groups;
	fbLightCtrl_Supl			: FB_LightSwitch;

	bTunningInProcess			: BOOL;
	bEnableLightCtrl			: BOOL;
	fbRTrigStartCtrl 			: R_TRIG;

//Tuning data
	fbPulsReadSensorData_TON	: TON;
	fbAutoTuneStartUpLevels		: FB_AutoTune_TcBA_Ex;
	fbR_TrigTuningDone			: R_TRIG ;
	fbStartStopLightCtrl: SR;
	
